LIN {X 0,Y 356.432,Z 513.307,A -85,B 0,C 180,E1 -13393.092,E2 -13393.092} C_VEL
LIN {X 0,Y 355.324,Z 522.171,A -85,B 0,C 180,E1 -13395.1,E2 -13395.1} C_VEL
LIN {X 0,Y 354.334,Z 530.476,A -85,B 0,C 180,E1 -13397.398,E2 -13397.398} C_VEL
LIN {X 0,Y 353.681,Z 537.111,A -85,B 0,C 180,E1 -13399.698,E2 -13399.698} C_VEL
LIN {X 0,Y 353.432,Z 542.27,A -85,B 0,C 180,E1 -13401.999,E2 -13401.999} C_VEL
LIN {X 0,Y 353.28,Z 546.062,A -85,B 0,C 180,E1 -13404.291,E2 -13404.291} C_VEL
LIN {X 0,Y 353.247,Z 548.565,A -85,B 0,C 180,E1 -13406.578,E2 -13406.578} C_VEL
LIN {X 0,Y 353.373,Z 549.83,A -85,B 0,C 180,E1 -13408.86,E2 -13408.86} C_VEL
LIN {X 0,Y 353.373,Z 549.828,A -85,B 0,C 180,E1 -13411.139,E2 -13411.139} C_VEL
LIN {X 0,Y 353.248,Z 548.554,A -85,B 0,C 180,E1 -13413.422,E2 -13413.422} C_VEL
LIN {X 0,Y 353.308,Z 546.046,A -85,B 0,C 180,E1 -13415.708,E2 -13415.708} C_VEL
LIN {X 0,Y 353.433,Z 542.253,A -85,B 0,C 180,E1 -13418.001,E2 -13418.001} C_VEL
LIN {X 0,Y 353.681,Z 537.089,A -85,B 0,C 180,E1 -13420.302,E2 -13420.302} C_VEL
LIN {X 0,Y 354.326,Z 530.439,A -85,B 0,C 180,E1 -13422.602,E2 -13422.602} C_VEL
LIN {X 0,Y 355.299,Z 522.123,A -85,B 0,C 180,E1 -13424.901,E2 -13424.901} C_VEL
LIN {X 0,Y 356.428,Z 513.256,A -85,B 0,C 180,E1 -13426.908,E2 -13426.908} C_VEL
LIN {X 0,Y 357.977,Z 502.598,A -85,B 0,C 180,E1 -13428.901,E2 -13428.901} C_VEL
LIN {X 0,Y 359.499,Z 491.658,A -85,B 0,C 180,E1 -13430.603,E2 -13430.603} C_VEL
LIN {X 0,Y 361.192,Z 479.725,A -85,B 0,C 180,E1 -13432.148,E2 -13432.148} C_VEL
LIN {X 0,Y 363.012,Z 466.679,A -85,B 0,C 180,E1 -13433.535,E2 -13433.535} C_VEL
LIN {X 0,Y 364.699,Z 454.014,A -85,B 0,C 180,E1 -13434.628,E2 -13434.628} C_VEL
LIN {X 0,Y 365.906,Z 442.133,A -85,B 0,C 180,E1 -13435.48,E2 -13435.48} C_VEL
LIN {X 0,Y 364.101,Z 428.944,A -85,B 0,C 180,E1 -13436.443,E2 -13436.443} C_VEL
LIN {X 0,Y 361.058,Z 413.785,A -85,B 0,C 180,E1 -13437.388,E2 -13437.388} C_VEL
LIN {X 0,Y 356.966,Z 398.611,A -85,B 0,C 180,E1 -13438.183,E2 -13438.183} C_VEL
LIN {X 0,Y 356.454,Z 396.29,A -85,B 0,C 180,E1 -13438.282,E2 -13438.282} C_VEL
LIN {X 0,Y 357.714,Z 387.602,A -85,B 0,C 180,E1 -13442.348,E2 -13442.348} C_VEL
LIN {X 0,Y 358.68,Z 381.362,A -85,B 0,C 180,E1 -13445.312,E2 -13445.312} C_VEL
LIN {X 0,Y 358.879,Z 378.763,A -85,B 0,C 180,E1 -13446.591,E2 -13446.591} C_VEL
LIN {X 0,Y 357.99,Z 373.352,A -85,B 0,C 180,E1 -13449.446,E2 -13449.446} C_VEL
LIN {X 0,Y 356.788,Z 366.727,A -85,B 0,C 180,E1 -13453.212,E2 -13453.212} C_VEL
LIN {X 0,Y 355.578,Z 360.645,A -85,B 0,C 180,E1 -13456.996,E2 -13456.996} C_VEL
LIN {X 0,Y 354.833,Z 356.903,A -85,B 0,C 180,E1 -13459.56,E2 -13459.56} C_VEL
LIN {X 0,Y 354.804,Z 356.919,A -85,B 0,C 180,E1 -13463.541,E2 -13463.541} C_VEL
LIN {X 0,Y 354.832,Z 356.914,A -85,B 0,C 180,E1 -13466.318,E2 -13466.318} C_VEL
LIN {X 0,Y 354.87,Z 356.908,A -85,B 0,C 180,E1 -13470.622,E2 -13470.622} C_VEL
LIN {X 0,Y 354.902,Z 356.902,A -85,B 0,C 180,E1 -13474.173,E2 -13474.173} C_VEL
LIN {X 0,Y 354.837,Z 356.912,A -85,B 0,C 180,E1 -13477.894,E2 -13477.894} C_VEL
LIN {X 0,Y 354.926,Z 356.897,A -85,B 0,C 180,E1 -13481.892,E2 -13481.892} C_VEL
LIN {X 0,Y 354.946,Z 356.896,A -85,B 0,C 180,E1 -13485.981,E2 -13485.981} C_VEL
LIN {X 0,Y 354.982,Z 356.889,A -85,B 0,C 180,E1 -13489.736,E2 -13489.736} C_VEL
LIN {X 0,Y 355.118,Z 356.871,A -85,B 0,C 180,E1 -13493.181,E2 -13493.181} C_VEL
LIN {X 0,Y 355.247,Z 356.854,A -85,B 0,C 180,E1 -13497.733,E2 -13497.733} C_VEL
LIN {X 0,Y 355.4,Z 356.836,A -85,B 0,C 180,E1 -13500,E2 -13500} C_VEL
LIN {X 0,Y 355.247,Z 356.859,A -85,B 0,C 180,E1 -13502.268,E2 -13502.268} C_VEL
LIN {X 0,Y 355.142,Z 356.87,A -85,B 0,C 180,E1 -13506.819,E2 -13506.819} C_VEL
LIN {X 0,Y 355.02,Z 356.886,A -85,B 0,C 180,E1 -13509.112,E2 -13509.112} C_VEL
LIN {X 0,Y 354.93,Z 356.897,A -85,B 0,C 180,E1 -13512.581,E2 -13512.581} C_VEL
LIN {X 0,Y 354.894,Z 356.902,A -85,B 0,C 180,E1 -13516.096,E2 -13516.096} C_VEL
LIN {X 0,Y 354.91,Z 356.898,A -85,B 0,C 180,E1 -13518.472,E2 -13518.472} C_VEL
LIN {X 0,Y 354.838,Z 356.911,A -85,B 0,C 180,E1 -13522.106,E2 -13522.106} C_VEL
LIN {X 0,Y 354.903,Z 356.901,A -85,B 0,C 180,E1 -13525.827,E2 -13525.827} C_VEL
LIN {X 0,Y 354.857,Z 356.904,A -85,B 0,C 180,E1 -13529.679,E2 -13529.679} C_VEL
LIN {X 0,Y 354.809,Z 356.915,A -85,B 0,C 180,E1 -13533.702,E2 -13533.702} C_VEL
LIN {X 0,Y 354.801,Z 356.916,A -85,B 0,C 180,E1 -13536.459,E2 -13536.459} C_VEL
LIN {X 0,Y 354.827,Z 356.913,A -85,B 0,C 180,E1 -13539.424,E2 -13539.424} C_VEL
LIN {X 0,Y 354.791,Z 356.916,A -85,B 0,C 180,E1 -13542.867,E2 -13542.867} C_VEL
LIN {X 0,Y 354.817,Z 357.055,A -85,B 0,C 180,E1 -13544.515,E2 -13544.515} C_VEL
LIN {X 0,Y 355.42,Z 360.567,A -85,B 0,C 180,E1 -13547.754,E2 -13547.754} C_VEL
LIN {X 0,Y 355.755,Z 364.073,A -85,B 0,C 180,E1 -13550.79,E2 -13550.79} C_VEL
LIN {X 0,Y 355.617,Z 367.534,A -85,B 0,C 180,E1 -13553.638,E2 -13553.638} C_VEL
LIN {X 0,Y 355.366,Z 371,A -85,B 0,C 180,E1 -13556.375,E2 -13556.375} C_VEL
LIN {X 0,Y 355.058,Z 374.488,A -85,B 0,C 180,E1 -13559.026,E2 -13559.026} C_VEL
LIN {X 0,Y 354.822,Z 378.006,A -85,B 0,C 180,E1 -13561.616,E2 -13561.616} C_VEL
LIN {X 0,Y 354.625,Z 381.777,A -85,B 0,C 180,E1 -13564.292,E2 -13564.292} C_VEL
LIN {X 0,Y 356.695,Z 387.842,A -85,B 0,C 180,E1 -13564.635,E2 -13564.635} C_VEL
LIN {X 0,Y 361.427,Z 402.417,A -85,B 0,C 180,E1 -13565.559,E2 -13565.559} C_VEL
LIN {X 0,Y 364.83,Z 415.964,A -85,B 0,C 180,E1 -13566.556,E2 -13566.556} C_VEL
LIN {X 0,Y 366.104,Z 422.295,A -85,B 0,C 180,E1 -13567.074,E2 -13567.074} C_VEL
LIN {X 0,Y 364.894,Z 435.031,A -85,B 0,C 180,E1 -13568.017,E2 -13568.017} C_VEL
LIN {X 0,Y 363.543,Z 446.261,A -85,B 0,C 180,E1 -13569.045,E2 -13569.045} C_VEL
LIN {X 0,Y 361.82,Z 458.433,A -85,B 0,C 180,E1 -13570.423,E2 -13570.423} C_VEL
LIN {X 0,Y 360.396,Z 468.475,A -85,B 0,C 180,E1 -13571.819,E2 -13571.819} C_VEL
LIN {X 0,Y 358.753,Z 478.455,A -85,B 0,C 180,E1 -13573.498,E2 -13573.498} C_VEL
LIN {X 0,Y 357.49,Z 486.727,A -85,B 0,C 180,E1 -13575.193,E2 -13575.193} C_VEL
LIN {X 0,Y 356.185,Z 494.631,A -85,B 0,C 180,E1 -13577.175,E2 -13577.175} C_VEL
LIN {X 0,Y 355.172,Z 501.015,A -85,B 0,C 180,E1 -13579.165,E2 -13579.165} C_VEL
LIN {X 0,Y 354.358,Z 506.684,A -85,B 0,C 180,E1 -13581.446,E2 -13581.446} C_VEL
LIN {X 0,Y 353.991,Z 509.96,A -85,B 0,C 180,E1 -13583.159,E2 -13583.159} C_VEL
LIN {X 0,Y 353.57,Z 513.105,A -85,B 0,C 180,E1 -13585.44,E2 -13585.44} C_VEL
LIN {X 0,Y 353.496,Z 514.951,A -85,B 0,C 180,E1 -13587.721,E2 -13587.721} C_VEL
LIN {X 0,Y 353.397,Z 515.581,A -85,B 0,C 180,E1 -13590,E2 -13590} C_VEL
LIN {X 0,Y 353.495,Z 515.006,A -85,B 0,C 180,E1 -13592.279,E2 -13592.279} C_VEL
LIN {X 0,Y 353.569,Z 513.22,A -85,B 0,C 180,E1 -13594.561,E2 -13594.561} C_VEL
LIN {X 0,Y 353.991,Z 510.136,A -85,B 0,C 180,E1 -13596.842,E2 -13596.842} C_VEL
LIN {X 0,Y 354.514,Z 505.659,A -85,B 0,C 180,E1 -13599.126,E2 -13599.126} C_VEL
LIN {X 0,Y 355.381,Z 499.628,A -85,B 0,C 180,E1 -13601.406,E2 -13601.406} C_VEL
LIN {X 0,Y 356.468,Z 492.907,A -85,B 0,C 180,E1 -13603.395,E2 -13603.395} C_VEL
LIN {X 0,Y 357.863,Z 484.866,A -85,B 0,C 180,E1 -13605.309,E2 -13605.309} C_VEL
LIN {X 0,Y 358.945,Z 477.477,A -85,B 0,C 180,E1 -13606.786,E2 -13606.786} C_VEL
LIN {X 0,Y 360.595,Z 467.25,A -85,B 0,C 180,E1 -13608.465,E2 -13608.465} C_VEL
LIN {X 0,Y 362.254,Z 455.812,A -85,B 0,C 180,E1 -13609.995,E2 -13609.995} C_VEL
LIN {X 0,Y 363.811,Z 444.405,A -85,B 0,C 180,E1 -13611.236,E2 -13611.236} C_VEL
LIN {X 0,Y 365.265,Z 431.504,A -85,B 0,C 180,E1 -13612.367,E2 -13612.367} C_VEL
LIN {X 0,Y 366.073,Z 421.795,A -85,B 0,C 180,E1 -13613.069,E2 -13613.069} C_VEL
LIN {X 0,Y 362.89,Z 407.718,A -85,B 0,C 180,E1 -13614.172,E2 -13614.172} C_VEL
LIN {X 0,Y 359.006,Z 394.651,A -85,B 0,C 180,E1 -13615.06,E2 -13615.06} C_VEL
LIN {X 0,Y 354.616,Z 381.77,A -85,B 0,C 180,E1 -13615.818,E2 -13615.818} C_VEL
LIN {X 0,Y 354.944,Z 376.407,A -85,B 0,C 180,E1 -13619.671,E2 -13619.671} C_VEL
LIN {X 0,Y 355.117,Z 374.097,A -85,B 0,C 180,E1 -13621.397,E2 -13621.397} C_VEL
LIN {X 0,Y 354.59,Z 372.967,A -85,B 0,C 180,E1 -13622.327,E2 -13622.327} C_VEL
LIN {X 0,Y 351.952,Z 371.428,A -85,B 0,C 180,E1 -13623.855,E2 -13623.855} C_VEL
LIN {X 0,Y 349.672,Z 370.256,A -85,B 0,C 180,E1 -13625.092,E2 -13625.092} C_VEL
LIN {X 0,Y 348.705,Z 369.259,A -85,B 0,C 180,E1 -13626.044,E2 -13626.044} C_VEL
LIN {X 0,Y 348.635,Z 368.886,A -85,B 0,C 180,E1 -13626.364,E2 -13626.364} C_VEL
LIN {X 0,Y 348.761,Z 366.131,A -85,B 0,C 180,E1 -13628.66,E2 -13628.66} C_VEL
LIN {X 0,Y 348.733,Z 364.408,A -85,B 0,C 180,E1 -13630.158,E2 -13630.158} C_VEL
LIN {X 0,Y 348.284,Z 360.78,A -85,B 0,C 180,E1 -13633.411,E2 -13633.411} C_VEL
LIN {X 0,Y 347.734,Z 357.793,A -85,B 0,C 180,E1 -13636.394,E2 -13636.394} C_VEL
LIN {X 0,Y 347.736,Z 357.792,A -85,B 0,C 180,E1 -13639.703,E2 -13639.703} C_VEL
LIN {X 0,Y 347.766,Z 357.79,A -85,B 0,C 180,E1 -13642.679,E2 -13642.679} C_VEL
LIN {X 0,Y 347.752,Z 357.791,A -85,B 0,C 180,E1 -13645.956,E2 -13645.956} C_VEL
LIN {X 0,Y 347.768,Z 357.79,A -85,B 0,C 180,E1 -13649.654,E2 -13649.654} C_VEL
LIN {X 0,Y 347.856,Z 357.78,A -85,B 0,C 180,E1 -13652.745,E2 -13652.745} C_VEL
LIN {X 0,Y 347.793,Z 357.786,A -85,B 0,C 180,E1 -13656.162,E2 -13656.162} C_VEL
LIN {X 0,Y 347.817,Z 357.783,A -85,B 0,C 180,E1 -13659.909,E2 -13659.909} C_VEL
LIN {X 0,Y 347.871,Z 357.775,A -85,B 0,C 180,E1 -13662.359,E2 -13662.359} C_VEL
LIN {X 0,Y 347.902,Z 357.773,A -85,B 0,C 180,E1 -13665.971,E2 -13665.971} C_VEL
LIN {X 0,Y 347.934,Z 357.77,A -85,B 0,C 180,E1 -13669.526,E2 -13669.526} C_VEL
LIN {X 0,Y 348.08,Z 357.748,A -85,B 0,C 180,E1 -13671.875,E2 -13671.875} C_VEL
LIN {X 0,Y 348.073,Z 357.75,A -85,B 0,C 180,E1 -13674.206,E2 -13674.206} C_VEL
LIN {X 0,Y 348.211,Z 357.732,A -85,B 0,C 180,E1 -13677.686,E2 -13677.686} C_VEL
LIN {X 0,Y 348.35,Z 357.72,A -85,B 0,C 180,E1 -13680,E2 -13680} C_VEL
LIN {X 0,Y 348.211,Z 357.735,A -85,B 0,C 180,E1 -13682.313,E2 -13682.313} C_VEL
LIN {X 0,Y 348.082,Z 357.751,A -85,B 0,C 180,E1 -13686.958,E2 -13686.958} C_VEL
LIN {X 0,Y 347.935,Z 357.768,A -85,B 0,C 180,E1 -13690.474,E2 -13690.474} C_VEL
LIN {X 0,Y 347.902,Z 357.774,A -85,B 0,C 180,E1 -13694.149,E2 -13694.149} C_VEL
LIN {X 0,Y 347.895,Z 357.78,A -85,B 0,C 180,E1 -13698.29,E2 -13698.29} C_VEL
LIN {X 0,Y 347.793,Z 357.793,A -85,B 0,C 180,E1 -13701.635,E2 -13701.635} C_VEL
LIN {X 0,Y 347.816,Z 357.784,A -85,B 0,C 180,E1 -13705.108,E2 -13705.108} C_VEL
LIN {X 0,Y 347.814,Z 357.786,A -85,B 0,C 180,E1 -13707.693,E2 -13707.693} C_VEL
LIN {X 0,Y 347.767,Z 357.79,A -85,B 0,C 180,E1 -13710.346,E2 -13710.346} C_VEL
LIN {X 0,Y 347.747,Z 357.795,A -85,B 0,C 180,E1 -13714.463,E2 -13714.463} C_VEL
LIN {X 0,Y 347.777,Z 357.793,A -85,B 0,C 180,E1 -13717.988,E2 -13717.988} C_VEL
LIN {X 0,Y 347.804,Z 357.927,A -85,B 0,C 180,E1 -13719.837,E2 -13719.837} C_VEL
LIN {X 0,Y 348.884,Z 363.299,A -85,B 0,C 180,E1 -13723.515,E2 -13723.515} C_VEL
LIN {X 0,Y 349.967,Z 368.768,A -85,B 0,C 180,E1 -13726.938,E2 -13726.938} C_VEL
LIN {X 0,Y 350.961,Z 374.276,A -85,B 0,C 180,E1 -13730.148,E2 -13730.148} C_VEL
LIN {X 0,Y 351.897,Z 379.829,A -85,B 0,C 180,E1 -13733.19,E2 -13733.19} C_VEL
LIN {X 0,Y 351.615,Z 383.488,A -85,B 0,C 180,E1 -13735.034,E2 -13735.034} C_VEL
LIN {X 0,Y 350.384,Z 390.794,A -85,B 0,C 180,E1 -13738.566,E2 -13738.566} C_VEL
LIN {X 0,Y 349.561,Z 396.09,A -85,B 0,C 180,E1 -13741.108,E2 -13741.108} C_VEL
LIN {X 0,Y 354.345,Z 414.03,A -85,B 0,C 180,E1 -13742.083,E2 -13742.083} C_VEL
LIN {X 0,Y 357.089,Z 427.45,A -85,B 0,C 180,E1 -13742.946,E2 -13742.946} C_VEL
LIN {X 0,Y 359.156,Z 441.19,A -85,B 0,C 180,E1 -13743.971,E2 -13743.971} C_VEL
LIN {X 0,Y 359.363,Z 442.934,A -85,B 0,C 180,E1 -13744.107,E2 -13744.107} C_VEL
LIN {X 0,Y 357.759,Z 457.127,A -85,B 0,C 180,E1 -13745.171,E2 -13745.171} C_VEL
LIN {X 0,Y 355.932,Z 470.571,A -85,B 0,C 180,E1 -13746.431,E2 -13746.431} C_VEL
LIN {X 0,Y 354.131,Z 482.904,A -85,B 0,C 180,E1 -13747.847,E2 -13747.847} C_VEL
LIN {X 0,Y 352.535,Z 492.979,A -85,B 0,C 180,E1 -13749.229,E2 -13749.229} C_VEL
LIN {X 0,Y 350.988,Z 503.92,A -85,B 0,C 180,E1 -13751.011,E2 -13751.011} C_VEL
LIN {X 0,Y 349.523,Z 512.923,A -85,B 0,C 180,E1 -13752.747,E2 -13752.747} C_VEL
LIN {X 0,Y 348.361,Z 521.799,A -85,B 0,C 180,E1 -13754.795,E2 -13754.795} C_VEL
LIN {X 0,Y 347.322,Z 530.113,A -85,B 0,C 180,E1 -13757.139,E2 -13757.139} C_VEL
LIN {X 0,Y 346.63,Z 536.754,A -85,B 0,C 180,E1 -13759.486,E2 -13759.486} C_VEL
LIN {X 0,Y 346.357,Z 541.918,A -85,B 0,C 180,E1 -13761.834,E2 -13761.834} C_VEL
LIN {X 0,Y 346.199,Z 545.714,A -85,B 0,C 180,E1 -13764.174,E2 -13764.174} C_VEL
LIN {X 0,Y 346.168,Z 548.22,A -85,B 0,C 180,E1 -13766.508,E2 -13766.508} C_VEL
LIN {X 0,Y 346.276,Z 549.485,A -85,B 0,C 180,E1 -13768.837,E2 -13768.837} C_VEL
LIN {X 0,Y 346.276,Z 549.482,A -85,B 0,C 180,E1 -13771.163,E2 -13771.163} C_VEL
LIN {X 0,Y 346.17,Z 548.208,A -85,B 0,C 180,E1 -13773.492,E2 -13773.492} C_VEL
LIN {X 0,Y 346.243,Z 545.52,A -85,B 0,C 180,E1 -13775.961,E2 -13775.961} C_VEL
LIN {X 0,Y 346.357,Z 541.9,A -85,B 0,C 180,E1 -13778.166,E2 -13778.166} C_VEL
LIN {X 0,Y 346.63,Z 536.73,A -85,B 0,C 180,E1 -13780.514,E2 -13780.514} C_VEL
LIN {X 0,Y 347.311,Z 530.073,A -85,B 0,C 180,E1 -13782.861,E2 -13782.861} C_VEL
LIN {X 0,Y 348.357,Z 521.749,A -85,B 0,C 180,E1 -13785.205,E2 -13785.205} C_VEL
LIN {X 0,Y 349.516,Z 512.868,A -85,B 0,C 180,E1 -13787.253,E2 -13787.253} C_VEL
LIN {X 0,Y 350.938,Z 503.85,A -85,B 0,C 180,E1 -13788.992,E2 -13788.992} C_VEL
LIN {X 0,Y 352.548,Z 492.92,A -85,B 0,C 180,E1 -13790.767,E2 -13790.767} C_VEL
LIN {X 0,Y 354.24,Z 481.636,A -85,B 0,C 180,E1 -13792.299,E2 -13792.299} C_VEL
LIN {X 0,Y 356.037,Z 469.04,A -85,B 0,C 180,E1 -13793.715,E2 -13793.715} C_VEL
LIN {X 0,Y 357.767,Z 456.972,A -85,B 0,C 180,E1 -13794.828,E2 -13794.828} C_VEL
LIN {X 0,Y 359.291,Z 443.142,A -85,B 0,C 180,E1 -13795.869,E2 -13795.869} C_VEL
LIN {X 0,Y 357.443,Z 429.698,A -85,B 0,C 180,E1 -13796.887,E2 -13796.887} C_VEL
LIN {X 0,Y 354.554,Z 414.95,A -85,B 0,C 180,E1 -13797.844,E2 -13797.844} C_VEL
LIN {X 0,Y 350.68,Z 400.439,A -85,B 0,C 180,E1 -13798.649,E2 -13798.649} C_VEL
LIN {X 0,Y 349.562,Z 396.051,A -85,B 0,C 180,E1 -13798.892,E2 -13798.892} C_VEL
LIN {X 0,Y 350.804,Z 388.028,A -85,B 0,C 180,E1 -13802.746,E2 -13802.746} C_VEL
LIN {X 0,Y 351.725,Z 382.545,A -85,B 0,C 180,E1 -13805.413,E2 -13805.413} C_VEL
LIN {X 0,Y 351.845,Z 379.503,A -85,B 0,C 180,E1 -13806.967,E2 -13806.967} C_VEL
LIN {X 0,Y 350.943,Z 374.198,A -85,B 0,C 180,E1 -13809.854,E2 -13809.854} C_VEL
LIN {X 0,Y 349.763,Z 367.681,A -85,B 0,C 180,E1 -13813.667,E2 -13813.667} C_VEL
LIN {X 0,Y 348.559,Z 361.667,A -85,B 0,C 180,E1 -13817.51,E2 -13817.51} C_VEL
LIN {X 0,Y 347.797,Z 357.79,A -85,B 0,C 180,E1 -13820.262,E2 -13820.262} C_VEL
LIN {X 0,Y 347.792,Z 357.793,A -85,B 0,C 180,E1 -13824.125,E2 -13824.125} C_VEL
LIN {X 0,Y 347.741,Z 357.797,A -85,B 0,C 180,E1 -13828.086,E2 -13828.086} C_VEL
LIN {X 0,Y 347.807,Z 357.789,A -85,B 0,C 180,E1 -13830.99,E2 -13830.99} C_VEL
LIN {X 0,Y 347.834,Z 357.784,A -85,B 0,C 180,E1 -13833.608,E2 -13833.608} C_VEL
LIN {X 0,Y 347.791,Z 357.787,A -85,B 0,C 180,E1 -13836.162,E2 -13836.162} C_VEL
LIN {X 0,Y 347.82,Z 357.786,A -85,B 0,C 180,E1 -13839.91,E2 -13839.91} C_VEL
LIN {X 0,Y 347.869,Z 357.776,A -85,B 0,C 180,E1 -13842.36,E2 -13842.36} C_VEL
LIN {X 0,Y 347.9,Z 357.774,A -85,B 0,C 180,E1 -13845.971,E2 -13845.971} C_VEL
LIN {X 0,Y 347.933,Z 357.769,A -85,B 0,C 180,E1 -13849.526,E2 -13849.526} C_VEL
LIN {X 0,Y 348.086,Z 357.748,A -85,B 0,C 180,E1 -13853.042,E2 -13853.042} C_VEL
LIN {X 0,Y 348.21,Z 357.731,A -85,B 0,C 180,E1 -13857.687,E2 -13857.687} C_VEL
LIN {X 0,Y 348.349,Z 357.714,A -85,B 0,C 180,E1 -13860,E2 -13860} C_VEL
LIN {X 0,Y 348.21,Z 357.736,A -85,B 0,C 180,E1 -13862.314,E2 -13862.314} C_VEL
LIN {X 0,Y 348.11,Z 357.745,A -85,B 0,C 180,E1 -13866.958,E2 -13866.958} C_VEL
LIN {X 0,Y 347.973,Z 357.764,A -85,B 0,C 180,E1 -13869.299,E2 -13869.299} C_VEL
LIN {X 0,Y 347.898,Z 357.774,A -85,B 0,C 180,E1 -13872.839,E2 -13872.839} C_VEL
LIN {X 0,Y 347.843,Z 357.782,A -85,B 0,C 180,E1 -13876.431,E2 -13876.431} C_VEL
LIN {X 0,Y 347.859,Z 357.779,A -85,B 0,C 180,E1 -13878.86,E2 -13878.86} C_VEL
LIN {X 0,Y 347.778,Z 357.789,A -85,B 0,C 180,E1 -13882.579,E2 -13882.579} C_VEL
LIN {X 0,Y 347.816,Z 357.784,A -85,B 0,C 180,E1 -13885.108,E2 -13885.108} C_VEL
LIN {X 0,Y 347.814,Z 357.783,A -85,B 0,C 180,E1 -13887.694,E2 -13887.694} C_VEL
LIN {X 0,Y 347.767,Z 357.79,A -85,B 0,C 180,E1 -13890.346,E2 -13890.346} C_VEL
LIN {X 0,Y 347.747,Z 357.794,A -85,B 0,C 180,E1 -13894.464,E2 -13894.464} C_VEL
LIN {X 0,Y 347.776,Z 357.79,A -85,B 0,C 180,E1 -13897.989,E2 -13897.989} C_VEL
LIN {X 0,Y 347.753,Z 357.793,A -85,B 0,C 180,E1 -13901.83,E2 -13901.83} C_VEL
LIN {X 0,Y 347.75,Z 357.918,A -85,B 0,C 180,E1 -13904.005,E2 -13904.005} C_VEL
LIN {X 0,Y 348.299,Z 360.743,A -85,B 0,C 180,E1 -13906.681,E2 -13906.681} C_VEL
LIN {X 0,Y 348.715,Z 364.377,A -85,B 0,C 180,E1 -13909.983,E2 -13909.983} C_VEL
LIN {X 0,Y 348.673,Z 367.707,A -85,B 0,C 180,E1 -13912.793,E2 -13912.793} C_VEL
LIN {X 0,Y 348.411,Z 371.417,A -85,B 0,C 180,E1 -13915.796,E2 -13915.796} C_VEL
LIN {X 0,Y 348.133,Z 374.692,A -85,B 0,C 180,E1 -13918.34,E2 -13918.34} C_VEL
LIN {X 0,Y 347.843,Z 378.22,A -85,B 0,C 180,E1 -13920.993,E2 -13920.993} C_VEL
LIN {X 0,Y 347.611,Z 381.993,A -85,B 0,C 180,E1 -13923.714,E2 -13923.714} C_VEL
LIN {X 0,Y 353.042,Z 397.77,A -85,B 0,C 180,E1 -13924.687,E2 -13924.687} C_VEL
LIN {X 0,Y 356.691,Z 410.649,A -85,B 0,C 180,E1 -13925.614,E2 -13925.614} C_VEL
LIN {X 0,Y 359.45,Z 423.04,A -85,B 0,C 180,E1 -13926.636,E2 -13926.636} C_VEL
LIN {X 0,Y 358.328,Z 435.735,A -85,B 0,C 180,E1 -13927.611,E2 -13927.611} C_VEL
LIN {X 0,Y 356.932,Z 446.729,A -85,B 0,C 180,E1 -13928.638,E2 -13928.638} C_VEL
LIN {X 0,Y 355.336,Z 457.783,A -85,B 0,C 180,E1 -13929.901,E2 -13929.901} C_VEL
LIN {X 0,Y 353.661,Z 468.878,A -85,B 0,C 180,E1 -13931.461,E2 -13931.461} C_VEL
LIN {X 0,Y 351.957,Z 478.84,A -85,B 0,C 180,E1 -13933.17,E2 -13933.17} C_VEL
LIN {X 0,Y 350.624,Z 487.1,A -85,B 0,C 180,E1 -13934.896,E2 -13934.896} C_VEL
LIN {X 0,Y 349.241,Z 494.996,A -85,B 0,C 180,E1 -13936.915,E2 -13936.915} C_VEL
LIN {X 0,Y 348.186,Z 501.372,A -85,B 0,C 180,E1 -13938.945,E2 -13938.945} C_VEL
LIN {X 0,Y 347.339,Z 507.036,A -85,B 0,C 180,E1 -13941.271,E2 -13941.271} C_VEL
LIN {X 0,Y 346.946,Z 510.311,A -85,B 0,C 180,E1 -13943.019,E2 -13943.019} C_VEL
LIN {X 0,Y 346.512,Z 513.452,A -85,B 0,C 180,E1 -13945.347,E2 -13945.347} C_VEL
LIN {X 0,Y 346.404,Z 515.297,A -85,B 0,C 180,E1 -13947.675,E2 -13947.675} C_VEL
LIN {X 0,Y 346.318,Z 515.925,A -85,B 0,C 180,E1 -13950,E2 -13950} C_VEL
LIN {X 0,Y 346.403,Z 515.352,A -85,B 0,C 180,E1 -13952.326,E2 -13952.326} C_VEL
LIN {X 0,Y 346.511,Z 513.565,A -85,B 0,C 180,E1 -13954.654,E2 -13954.654} C_VEL
LIN {X 0,Y 346.946,Z 510.484,A -85,B 0,C 180,E1 -13956.981,E2 -13956.981} C_VEL
LIN {X 0,Y 347.502,Z 506.011,A -85,B 0,C 180,E1 -13959.311,E2 -13959.311} C_VEL
LIN {X 0,Y 348.419,Z 499.985,A -85,B 0,C 180,E1 -13961.637,E2 -13961.637} C_VEL
LIN {X 0,Y 349.552,Z 493.272,A -85,B 0,C 180,E1 -13963.665,E2 -13963.665} C_VEL
LIN {X 0,Y 350.976,Z 485.438,A -85,B 0,C 180,E1 -13965.572,E2 -13965.572} C_VEL
LIN {X 0,Y 352.138,Z 477.863,A -85,B 0,C 180,E1 -13967.121,E2 -13967.121} C_VEL
LIN {X 0,Y 353.887,Z 467.657,A -85,B 0,C 180,E1 -13968.828,E2 -13968.828} C_VEL
LIN {X 0,Y 355.424,Z 457.419,A -85,B 0,C 180,E1 -13970.245,E2 -13970.245} C_VEL
LIN {X 0,Y 357.055,Z 446.3,A -85,B 0,C 180,E1 -13971.506,E2 -13971.506} C_VEL
LIN {X 0,Y 358.532,Z 433.687,A -85,B 0,C 180,E1 -13972.67,E2 -13972.67} C_VEL
LIN {X 0,Y 359.568,Z 423.86,A -85,B 0,C 180,E1 -13973.397,E2 -13973.397} C_VEL
LIN {X 0,Y 356.919,Z 411.45,A -85,B 0,C 180,E1 -13974.426,E2 -13974.426} C_VEL
LIN {X 0,Y 353.318,Z 398.651,A -85,B 0,C 180,E1 -13975.359,E2 -13975.359} C_VEL
LIN {X 0,Y 348.541,Z 384.929,A -85,B 0,C 180,E1 -13976.23,E2 -13976.23} C_VEL
LIN {X 0,Y 347.619,Z 381.964,A -85,B 0,C 180,E1 -13976.41,E2 -13976.41} C_VEL
LIN {X 0,Y 347.976,Z 376.617,A -85,B 0,C 180,E1 -13980.326,E2 -13980.326} C_VEL
LIN {X 0,Y 348.262,Z 373.108,A -85,B 0,C 180,E1 -13983.016,E2 -13983.016} C_VEL
LIN {X 0,Y 348.635,Z 368.886,A -85,B 0,C 180,E1 -13986.364,E2 -13986.364} C_VEL
LIN {X 0,Y 348.009,Z 367.867,A -85,B 0,C 180,E1 -13987.315,E2 -13987.315} C_VEL
LIN {X 0,Y 345.216,Z 366.529,A -85,B 0,C 180,E1 -13988.873,E2 -13988.873} C_VEL
LIN {X 0,Y 342.788,Z 365.501,A -85,B 0,C 180,E1 -13990.134,E2 -13990.134} C_VEL
LIN {X 0,Y 341.677,Z 364.596,A -85,B 0,C 180,E1 -13991.107,E2 -13991.107} C_VEL
LIN {X 0,Y 341.55,Z 364.255,A -85,B 0,C 180,E1 -13991.435,E2 -13991.435} C_VEL
LIN {X 0,Y 341.07,Z 361,A -85,B 0,C 180,E1 -13994.475,E2 -13994.475} C_VEL
LIN {X 0,Y 340.68,Z 358.671,A -85,B 0,C 180,E1 -13996.87,E2 -13996.87} C_VEL
LIN {X 0,Y 340.703,Z 358.668,A -85,B 0,C 180,E1 -14000.248,E2 -14000.248} C_VEL
LIN {X 0,Y 340.714,Z 358.669,A -85,B 0,C 180,E1 -14003.559,E2 -14003.559} C_VEL
LIN {X 0,Y 340.696,Z 358.671,A -85,B 0,C 180,E1 -14006.154,E2 -14006.154} C_VEL
LIN {X 0,Y 340.779,Z 358.663,A -85,B 0,C 180,E1 -14010.333,E2 -14010.333} C_VEL
LIN {X 0,Y 340.809,Z 358.66,A -85,B 0,C 180,E1 -14013.02,E2 -14013.02} C_VEL
LIN {X 0,Y 340.761,Z 358.663,A -85,B 0,C 180,E1 -14015.638,E2 -14015.638} C_VEL
LIN {X 0,Y 340.75,Z 358.66,A -85,B 0,C 180,E1 -14019.474,E2 -14019.474} C_VEL
LIN {X 0,Y 340.862,Z 358.647,A -85,B 0,C 180,E1 -14021.984,E2 -14021.984} C_VEL
LIN {X 0,Y 340.874,Z 358.648,A -85,B 0,C 180,E1 -14025.705,E2 -14025.705} C_VEL
LIN {X 0,Y 340.876,Z 358.648,A -85,B 0,C 180,E1 -14029.306,E2 -14029.306} C_VEL
LIN {X 0,Y 341.081,Z 358.623,A -85,B 0,C 180,E1 -14032.898,E2 -14032.898} C_VEL
LIN {X 0,Y 341.173,Z 358.609,A -85,B 0,C 180,E1 -14037.639,E2 -14037.639} C_VEL
LIN {X 0,Y 341.3,Z 358.598,A -85,B 0,C 180,E1 -14040,E2 -14040} C_VEL
LIN {X 0,Y 341.173,Z 358.612,A -85,B 0,C 180,E1 -14042.361,E2 -14042.361} C_VEL
LIN {X 0,Y 341.05,Z 358.626,A -85,B 0,C 180,E1 -14047.102,E2 -14047.102} C_VEL
LIN {X 0,Y 340.878,Z 358.646,A -85,B 0,C 180,E1 -14050.693,E2 -14050.693} C_VEL
LIN {X 0,Y 340.867,Z 358.65,A -85,B 0,C 180,E1 -14054.324,E2 -14054.324} C_VEL
LIN {X 0,Y 340.842,Z 358.66,A -85,B 0,C 180,E1 -14058.467,E2 -14058.467} C_VEL
LIN {X 0,Y 340.757,Z 358.667,A -85,B 0,C 180,E1 -14061.856,E2 -14061.856} C_VEL
LIN {X 0,Y 340.776,Z 358.661,A -85,B 0,C 180,E1 -14065.664,E2 -14065.664} C_VEL
LIN {X 0,Y 340.744,Z 358.667,A -85,B 0,C 180,E1 -14068.319,E2 -14068.319} C_VEL
LIN {X 0,Y 340.707,Z 358.673,A -85,B 0,C 180,E1 -14071.044,E2 -14071.044} C_VEL
LIN {X 0,Y 340.721,Z 358.675,A -85,B 0,C 180,E1 -14075.278,E2 -14075.278} C_VEL
LIN {X 0,Y 340.729,Z 358.706,A -85,B 0,C 180,E1 -14079.013,E2 -14079.013} C_VEL
LIN {X 0,Y 341.794,Z 363.925,A -85,B 0,C 180,E1 -14082.73,E2 -14082.73} C_VEL
LIN {X 0,Y 342.74,Z 368.716,A -85,B 0,C 180,E1 -14085.864,E2 -14085.864} C_VEL
LIN {X 0,Y 343.732,Z 374.131,A -85,B 0,C 180,E1 -14089.157,E2 -14089.157} C_VEL
LIN {X 0,Y 344.815,Z 380.267,A -85,B 0,C 180,E1 -14092.645,E2 -14092.645} C_VEL
LIN {X 0,Y 344.942,Z 382.387,A -85,B 0,C 180,E1 -14093.782,E2 -14093.782} C_VEL
LIN {X 0,Y 343.915,Z 388.618,A -85,B 0,C 180,E1 -14096.913,E2 -14096.913} C_VEL
LIN {X 0,Y 342.719,Z 395.923,A -85,B 0,C 180,E1 -14100.517,E2 -14100.517} C_VEL
LIN {X 0,Y 347.509,Z 413.681,A -85,B 0,C 180,E1 -14101.511,E2 -14101.511} C_VEL
LIN {X 0,Y 350.429,Z 427.822,A -85,B 0,C 180,E1 -14102.45,E2 -14102.45} C_VEL
LIN {X 0,Y 352.491,Z 441.872,A -85,B 0,C 180,E1 -14103.534,E2 -14103.534} C_VEL
LIN {X 0,Y 352.606,Z 445.116,A -85,B 0,C 180,E1 -14103.792,E2 -14103.792} C_VEL
LIN {X 0,Y 351.055,Z 458.246,A -85,B 0,C 180,E1 -14104.825,E2 -14104.825} C_VEL
LIN {X 0,Y 349.175,Z 471.414,A -85,B 0,C 180,E1 -14106.104,E2 -14106.104} C_VEL
LIN {X 0,Y 347.326,Z 483.574,A -85,B 0,C 180,E1 -14107.547,E2 -14107.547} C_VEL
LIN {X 0,Y 345.613,Z 494.023,A -85,B 0,C 180,E1 -14109.024,E2 -14109.024} C_VEL
LIN {X 0,Y 343.946,Z 505.175,A -85,B 0,C 180,E1 -14110.917,E2 -14110.917} C_VEL
LIN {X 0,Y 342.269,Z 515.293,A -85,B 0,C 180,E1 -14112.986,E2 -14112.986} C_VEL
LIN {X 0,Y 341.149,Z 523.721,A -85,B 0,C 180,E1 -14115.077,E2 -14115.077} C_VEL
LIN {X 0,Y 340.145,Z 531.602,A -85,B 0,C 180,E1 -14117.47,E2 -14117.47} C_VEL
LIN {X 0,Y 339.477,Z 537.861,A -85,B 0,C 180,E1 -14119.865,E2 -14119.865} C_VEL
LIN {X 0,Y 339.218,Z 542.677,A -85,B 0,C 180,E1 -14122.26,E2 -14122.26} C_VEL
LIN {X 0,Y 339.128,Z 545.451,A -85,B 0,C 180,E1 -14124.118,E2 -14124.118} C_VEL
LIN {X 0,Y 339.092,Z 547.874,A -85,B 0,C 180,E1 -14126.435,E2 -14126.435} C_VEL
LIN {X 0,Y 339.179,Z 549.139,A -85,B 0,C 180,E1 -14128.813,E2 -14128.813} C_VEL
LIN {X 0,Y 339.222,Z 549.303,A -85,B 0,C 180,E1 -14130,E2 -14130} C_VEL
LIN {X 0,Y 339.09,Z 548.652,A -85,B 0,C 180,E1 -14132.376,E2 -14132.376} C_VEL
LIN {X 0,Y 339.127,Z 546.763,A -85,B 0,C 180,E1 -14134.755,E2 -14134.755} C_VEL
LIN {X 0,Y 339.222,Z 543.614,A -85,B 0,C 180,E1 -14137.141,E2 -14137.141} C_VEL
LIN {X 0,Y 339.394,Z 539.137,A -85,B 0,C 180,E1 -14139.536,E2 -14139.536} C_VEL
LIN {X 0,Y 339.962,Z 533.238,A -85,B 0,C 180,E1 -14141.931,E2 -14141.931} C_VEL
LIN {X 0,Y 340.783,Z 525.762,A -85,B 0,C 180,E1 -14144.328,E2 -14144.328} C_VEL
LIN {X 0,Y 341.893,Z 517.762,A -85,B 0,C 180,E1 -14146.418,E2 -14146.418} C_VEL
LIN {X 0,Y 343.427,Z 508.15,A -85,B 0,C 180,E1 -14148.494,E2 -14148.494} C_VEL
LIN {X 0,Y 344.967,Z 498.35,A -85,B 0,C 180,E1 -14150.264,E2 -14150.264} C_VEL
LIN {X 0,Y 346.714,Z 486.705,A -85,B 0,C 180,E1 -14152.024,E2 -14152.024} C_VEL
LIN {X 0,Y 348.746,Z 473.884,A -85,B 0,C 180,E1 -14153.611,E2 -14153.611} C_VEL
LIN {X 0,Y 350.58,Z 461.209,A -85,B 0,C 180,E1 -14154.897,E2 -14154.897} C_VEL
LIN {X 0,Y 352.324,Z 447.392,A -85,B 0,C 180,E1 -14156.03,E2 -14156.03} C_VEL
LIN {X 0,Y 352.71,Z 443.953,A -85,B 0,C 180,E1 -14156.278,E2 -14156.278} C_VEL
LIN {X 0,Y 350.89,Z 430.908,A -85,B 0,C 180,E1 -14157.311,E2 -14157.311} C_VEL
LIN {X 0,Y 348.227,Z 416.81,A -85,B 0,C 180,E1 -14158.271,E2 -14158.271} C_VEL
LIN {X 0,Y 344.357,Z 401.886,A -85,B 0,C 180,E1 -14159.147,E2 -14159.147} C_VEL
LIN {X 0,Y 342.713,Z 395.88,A -85,B 0,C 180,E1 -14159.483,E2 -14159.483} C_VEL
LIN {X 0,Y 343.913,Z 388.583,A -85,B 0,C 180,E1 -14163.086,E2 -14163.086} C_VEL
LIN {X 0,Y 344.915,Z 382.337,A -85,B 0,C 180,E1 -14166.221,E2 -14166.221} C_VEL
LIN {X 0,Y 344.54,Z 378.324,A -85,B 0,C 180,E1 -14168.407,E2 -14168.407} C_VEL
LIN {X 0,Y 343.195,Z 371.255,A -85,B 0,C 180,E1 -14172.515,E2 -14172.515} C_VEL
LIN {X 0,Y 342.13,Z 365.788,A -85,B 0,C 180,E1 -14175.97,E2 -14175.97} C_VEL
LIN {X 0,Y 341.104,Z 360.436,A -85,B 0,C 180,E1 -14179.671,E2 -14179.671} C_VEL
LIN {X 0,Y 340.738,Z 358.669,A -85,B 0,C 180,E1 -14180.986,E2 -14180.986} C_VEL
LIN {X 0,Y 340.72,Z 358.675,A -85,B 0,C 180,E1 -14184.722,E2 -14184.722} C_VEL
LIN {X 0,Y 340.706,Z 358.675,A -85,B 0,C 180,E1 -14188.956,E2 -14188.956} C_VEL
LIN {X 0,Y 340.781,Z 358.661,A -85,B 0,C 180,E1 -14192.474,E2 -14192.474} C_VEL
LIN {X 0,Y 340.758,Z 358.665,A -85,B 0,C 180,E1 -14195.639,E2 -14195.639} C_VEL
LIN {X 0,Y 340.751,Z 358.662,A -85,B 0,C 180,E1 -14199.475,E2 -14199.475} C_VEL
LIN {X 0,Y 340.861,Z 358.649,A -85,B 0,C 180,E1 -14201.985,E2 -14201.985} C_VEL
LIN {X 0,Y 340.872,Z 358.649,A -85,B 0,C 180,E1 -14205.705,E2 -14205.705} C_VEL
LIN {X 0,Y 340.876,Z 358.649,A -85,B 0,C 180,E1 -14209.307,E2 -14209.307} C_VEL
LIN {X 0,Y 341.053,Z 358.625,A -85,B 0,C 180,E1 -14212.898,E2 -14212.898} C_VEL
LIN {X 0,Y 341.171,Z 358.607,A -85,B 0,C 180,E1 -14217.639,E2 -14217.639} C_VEL
LIN {X 0,Y 341.299,Z 358.592,A -85,B 0,C 180,E1 -14220,E2 -14220} C_VEL
LIN {X 0,Y 341.171,Z 358.612,A -85,B 0,C 180,E1 -14222.361,E2 -14222.361} C_VEL
LIN {X 0,Y 341.08,Z 358.62,A -85,B 0,C 180,E1 -14227.102,E2 -14227.102} C_VEL
LIN {X 0,Y 340.879,Z 358.646,A -85,B 0,C 180,E1 -14230.694,E2 -14230.694} C_VEL
LIN {X 0,Y 340.866,Z 358.648,A -85,B 0,C 180,E1 -14234.325,E2 -14234.325} C_VEL
LIN {X 0,Y 340.841,Z 358.65,A -85,B 0,C 180,E1 -14238.467,E2 -14238.467} C_VEL
LIN {X 0,Y 340.757,Z 358.662,A -85,B 0,C 180,E1 -14241.857,E2 -14241.857} C_VEL
LIN {X 0,Y 340.776,Z 358.661,A -85,B 0,C 180,E1 -14245.664,E2 -14245.664} C_VEL
LIN {X 0,Y 340.744,Z 358.667,A -85,B 0,C 180,E1 -14248.32,E2 -14248.32} C_VEL
LIN {X 0,Y 340.707,Z 358.67,A -85,B 0,C 180,E1 -14251.044,E2 -14251.044} C_VEL
LIN {X 0,Y 340.721,Z 358.671,A -85,B 0,C 180,E1 -14255.279,E2 -14255.279} C_VEL
LIN {X 0,Y 340.712,Z 358.669,A -85,B 0,C 180,E1 -14258.386,E2 -14258.386} C_VEL
LIN {X 0,Y 340.701,Z 358.673,A -85,B 0,C 180,E1 -14262.046,E2 -14262.046} C_VEL
LIN {X 0,Y 340.713,Z 358.819,A -85,B 0,C 180,E1 -14263.511,E2 -14263.511} C_VEL
LIN {X 0,Y 341.194,Z 361.508,A -85,B 0,C 180,E1 -14266.132,E2 -14266.132} C_VEL
LIN {X 0,Y 341.686,Z 365.209,A -85,B 0,C 180,E1 -14269.556,E2 -14269.556} C_VEL
LIN {X 0,Y 341.731,Z 367.878,A -85,B 0,C 180,E1 -14271.904,E2 -14271.904} C_VEL
LIN {X 0,Y 341.431,Z 372.128,A -85,B 0,C 180,E1 -14275.423,E2 -14275.423} C_VEL
LIN {X 0,Y 341.013,Z 376.658,A -85,B 0,C 180,E1 -14278.987,E2 -14278.987} C_VEL
LIN {X 0,Y 340.685,Z 381.346,A -85,B 0,C 180,E1 -14282.505,E2 -14282.505} C_VEL
LIN {X 0,Y 340.655,Z 382.153,A -85,B 0,C 180,E1 -14283.099,E2 -14283.099} C_VEL
LIN {X 0,Y 341.735,Z 385.452,A -85,B 0,C 180,E1 -14283.291,E2 -14283.291} C_VEL
LIN {X 0,Y 346.616,Z 399.446,A -85,B 0,C 180,E1 -14284.217,E2 -14284.217} C_VEL
LIN {X 0,Y 350.183,Z 412.204,A -85,B 0,C 180,E1 -14285.182,E2 -14285.182} C_VEL
LIN {X 0,Y 352.749,Z 423.844,A -85,B 0,C 180,E1 -14286.181,E2 -14286.181} C_VEL
LIN {X 0,Y 352.771,Z 426.742,A -85,B 0,C 180,E1 -14286.409,E2 -14286.409} C_VEL
LIN {X 0,Y 351.3,Z 440.313,A -85,B 0,C 180,E1 -14287.534,E2 -14287.534} C_VEL
LIN {X 0,Y 349.693,Z 452.352,A -85,B 0,C 180,E1 -14288.792,E2 -14288.792} C_VEL
LIN {X 0,Y 347.88,Z 463.525,A -85,B 0,C 180,E1 -14290.221,E2 -14290.221} C_VEL
LIN {X 0,Y 346.019,Z 474.488,A -85,B 0,C 180,E1 -14291.956,E2 -14291.956} C_VEL
LIN {X 0,Y 344.365,Z 483.752,A -85,B 0,C 180,E1 -14293.753,E2 -14293.753} C_VEL
LIN {X 0,Y 342.94,Z 492.164,A -85,B 0,C 180,E1 -14295.764,E2 -14295.764} C_VEL
LIN {X 0,Y 341.851,Z 498.276,A -85,B 0,C 180,E1 -14297.534,E2 -14297.534} C_VEL
LIN {X 0,Y 340.735,Z 504.755,A -85,B 0,C 180,E1 -14299.903,E2 -14299.903} C_VEL
LIN {X 0,Y 340.013,Z 509.643,A -85,B 0,C 180,E1 -14302.279,E2 -14302.279} C_VEL
LIN {X 0,Y 339.68,Z 512.395,A -85,B 0,C 180,E1 -14304.062,E2 -14304.062} C_VEL
LIN {X 0,Y 339.328,Z 514.879,A -85,B 0,C 180,E1 -14306.438,E2 -14306.438} C_VEL
LIN {X 0,Y 339.274,Z 516.107,A -85,B 0,C 180,E1 -14308.813,E2 -14308.813} C_VEL
LIN {X 0,Y 339.274,Z 516.133,A -85,B 0,C 180,E1 -14311.187,E2 -14311.187} C_VEL
LIN {X 0,Y 339.327,Z 514.961,A -85,B 0,C 180,E1 -14313.563,E2 -14313.563} C_VEL
LIN {X 0,Y 339.679,Z 512.536,A -85,B 0,C 180,E1 -14315.938,E2 -14315.938} C_VEL
LIN {X 0,Y 340.147,Z 508.782,A -85,B 0,C 180,E1 -14318.316,E2 -14318.316} C_VEL
LIN {X 0,Y 340.949,Z 503.557,A -85,B 0,C 180,E1 -14320.692,E2 -14320.692} C_VEL
LIN {X 0,Y 342.071,Z 496.685,A -85,B 0,C 180,E1 -14323.062,E2 -14323.062} C_VEL
LIN {X 0,Y 343.542,Z 489.09,A -85,B 0,C 180,E1 -14325.12,E2 -14325.12} C_VEL
LIN {X 0,Y 344.863,Z 481.184,A -85,B 0,C 180,E1 -14326.882,E2 -14326.882} C_VEL
LIN {X 0,Y 346.543,Z 471.648,A -85,B 0,C 180,E1 -14328.628,E2 -14328.628} C_VEL
LIN {X 0,Y 348.275,Z 461.067,A -85,B 0,C 180,E1 -14330.217,E2 -14330.217} C_VEL
LIN {X 0,Y 350.102,Z 449.355,A -85,B 0,C 180,E1 -14331.646,E2 -14331.646} C_VEL
LIN {X 0,Y 351.745,Z 436.776,A -85,B 0,C 180,E1 -14332.886,E2 -14332.886} C_VEL
LIN {X 0,Y 352.93,Z 424.653,A -85,B 0,C 180,E1 -14333.848,E2 -14333.848} C_VEL
LIN {X 0,Y 350.239,Z 412.156,A -85,B 0,C 180,E1 -14334.923,E2 -14334.923} C_VEL
LIN {X 0,Y 346.503,Z 398.991,A -85,B 0,C 180,E1 -14335.92,E2 -14335.92} C_VEL
LIN {X 0,Y 341.671,Z 385.294,A -85,B 0,C 180,E1 -14336.828,E2 -14336.828} C_VEL
LIN {X 0,Y 340.657,Z 382.132,A -85,B 0,C 180,E1 -14337.024,E2 -14337.024} C_VEL
LIN {X 0,Y 340.938,Z 378.092,A -85,B 0,C 180,E1 -14340.028,E2 -14340.028} C_VEL
LIN {X 0,Y 341.326,Z 373.3,A -85,B 0,C 180,E1 -14343.776,E2 -14343.776} C_VEL
LIN {X 0,Y 341.672,Z 369.733,A -85,B 0,C 180,E1 -14346.658,E2 -14346.658} C_VEL
LIN {X 0,Y 341.761,Z 366.302,A -85,B 0,C 180,E1 -14349.605,E2 -14349.605} C_VEL
LIN {X 0,Y 341.55,Z 364.255,A -85,B 0,C 180,E1 -14351.435,E2 -14351.435} C_VEL
LIN {X 0,Y 340.746,Z 363.346,A -85,B 0,C 180,E1 -14352.405,E2 -14352.405} C_VEL
LIN {X 0,Y 337.676,Z 362.218,A -85,B 0,C 180,E1 -14353.985,E2 -14353.985} C_VEL
LIN {X 0,Y 335.078,Z 361.372,A -85,B 0,C 180,E1 -14355.266,E2 -14355.266} C_VEL
LIN {X 0,Y 333.888,Z 360.581,A -85,B 0,C 180,E1 -14356.257,E2 -14356.257} C_VEL
LIN {X 0,Y 333.749,Z 360.266,A -85,B 0,C 180,E1 -14356.593,E2 -14356.593} C_VEL
LIN {X 0,Y 333.644,Z 359.547,A -85,B 0,C 180,E1 -14357.618,E2 -14357.618} C_VEL
LIN {X 0,Y 333.656,Z 359.546,A -85,B 0,C 180,E1 -14361.202,E2 -14361.202} C_VEL
LIN {X 0,Y 333.68,Z 359.545,A -85,B 0,C 180,E1 -14363.861,E2 -14363.861} C_VEL
LIN {X 0,Y 333.647,Z 359.549,A -85,B 0,C 180,E1 -14367.413,E2 -14367.413} C_VEL
LIN {X 0,Y 333.715,Z 359.542,A -85,B 0,C 180,E1 -14371.028,E2 -14371.028} C_VEL
LIN {X 0,Y 333.74,Z 359.535,A -85,B 0,C 180,E1 -14373.754,E2 -14373.754} C_VEL
LIN {X 0,Y 333.724,Z 359.541,A -85,B 0,C 180,E1 -14377.914,E2 -14377.914} C_VEL
LIN {X 0,Y 333.798,Z 359.528,A -85,B 0,C 180,E1 -14381.589,E2 -14381.589} C_VEL
LIN {X 0,Y 333.813,Z 359.527,A -85,B 0,C 180,E1 -14385.576,E2 -14385.576} C_VEL
LIN {X 0,Y 333.839,Z 359.525,A -85,B 0,C 180,E1 -14389.078,E2 -14389.078} C_VEL
LIN {X 0,Y 334.031,Z 359.501,A -85,B 0,C 180,E1 -14392.747,E2 -14392.747} C_VEL
LIN {X 0,Y 333.815,Z 359.524,A -85,B 0,C 180,E1 -14395.169,E2 -14395.169} C_VEL
LIN {X 0,Y 334.11,Z 359.489,A -85,B 0,C 180,E1 -14397.589,E2 -14397.589} C_VEL
LIN {X 0,Y 334.251,Z 359.477,A -85,B 0,C 180,E1 -14400,E2 -14400} C_VEL
LIN {X 0,Y 334.11,Z 359.492,A -85,B 0,C 180,E1 -14402.411,E2 -14402.411} C_VEL
LIN {X 0,Y 334.013,Z 359.504,A -85,B 0,C 180,E1 -14406.039,E2 -14406.039} C_VEL
LIN {X 0,Y 333.854,Z 359.526,A -85,B 0,C 180,E1 -14409.695,E2 -14409.695} C_VEL
LIN {X 0,Y 333.803,Z 359.532,A -85,B 0,C 180,E1 -14413.391,E2 -14413.391} C_VEL
LIN {X 0,Y 333.751,Z 359.538,A -85,B 0,C 180,E1 -14417.146,E2 -14417.146} C_VEL
LIN {X 0,Y 333.746,Z 359.538,A -85,B 0,C 180,E1 -14419.69,E2 -14419.69} C_VEL
LIN {X 0,Y 333.696,Z 359.543,A -85,B 0,C 180,E1 -14422.278,E2 -14422.278} C_VEL
LIN {X 0,Y 333.739,Z 359.54,A -85,B 0,C 180,E1 -14426.246,E2 -14426.246} C_VEL
LIN {X 0,Y 333.714,Z 359.543,A -85,B 0,C 180,E1 -14428.972,E2 -14428.972} C_VEL
LIN {X 0,Y 333.648,Z 359.551,A -85,B 0,C 180,E1 -14432.587,E2 -14432.587} C_VEL
LIN {X 0,Y 333.679,Z 359.551,A -85,B 0,C 180,E1 -14436.138,E2 -14436.138} C_VEL
LIN {X 0,Y 333.716,Z 359.598,A -85,B 0,C 180,E1 -14438.248,E2 -14438.248} C_VEL
LIN {X 0,Y 334.769,Z 364.961,A -85,B 0,C 180,E1 -14442.206,E2 -14442.206} C_VEL
LIN {X 0,Y 335.714,Z 369.642,A -85,B 0,C 180,E1 -14445.379,E2 -14445.379} C_VEL
LIN {X 0,Y 336.677,Z 374.979,A -85,B 0,C 180,E1 -14448.719,E2 -14448.719} C_VEL
LIN {X 0,Y 337.766,Z 381.018,A -85,B 0,C 180,E1 -14452.249,E2 -14452.249} C_VEL
LIN {X 0,Y 337.852,Z 384.61,A -85,B 0,C 180,E1 -14454.221,E2 -14454.221} C_VEL
LIN {X 0,Y 336.595,Z 391.689,A -85,B 0,C 180,E1 -14457.83,E2 -14457.83} C_VEL
LIN {X 0,Y 335.873,Z 395.952,A -85,B 0,C 180,E1 -14459.91,E2 -14459.91} C_VEL
LIN {X 0,Y 340.314,Z 411.998,A -85,B 0,C 180,E1 -14460.829,E2 -14460.829} C_VEL
LIN {X 0,Y 343.522,Z 426.734,A -85,B 0,C 180,E1 -14461.832,E2 -14461.832} C_VEL
LIN {X 0,Y 345.671,Z 441.133,A -85,B 0,C 180,E1 -14462.963,E2 -14462.963} C_VEL
LIN {X 0,Y 346.023,Z 446.004,A -85,B 0,C 180,E1 -14463.375,E2 -14463.375} C_VEL
LIN {X 0,Y 344.361,Z 459.458,A -85,B 0,C 180,E1 -14464.477,E2 -14464.477} C_VEL
LIN {X 0,Y 342.413,Z 472.25,A -85,B 0,C 180,E1 -14465.763,E2 -14465.763} C_VEL
LIN {X 0,Y 340.519,Z 484.225,A -85,B 0,C 180,E1 -14467.233,E2 -14467.233} C_VEL
LIN {X 0,Y 338.734,Z 494.778,A -85,B 0,C 180,E1 -14468.774,E2 -14468.774} C_VEL
LIN {X 0,Y 337.166,Z 504.783,A -85,B 0,C 180,E1 -14470.518,E2 -14470.518} C_VEL
LIN {X 0,Y 335.4,Z 514.917,A -85,B 0,C 180,E1 -14472.626,E2 -14472.626} C_VEL
LIN {X 0,Y 334.179,Z 523.35,A -85,B 0,C 180,E1 -14474.759,E2 -14474.759} C_VEL
LIN {X 0,Y 333.32,Z 529.388,A -85,B 0,C 180,E1 -14476.589,E2 -14476.589} C_VEL
LIN {X 0,Y 332.543,Z 536.041,A -85,B 0,C 180,E1 -14479.035,E2 -14479.035} C_VEL
LIN {X 0,Y 332.212,Z 541.214,A -85,B 0,C 180,E1 -14481.484,E2 -14481.484} C_VEL
LIN {X 0,Y 332.04,Z 545.018,A -85,B 0,C 180,E1 -14483.925,E2 -14483.925} C_VEL
LIN {X 0,Y 332.016,Z 547.529,A -85,B 0,C 180,E1 -14486.359,E2 -14486.359} C_VEL
LIN {X 0,Y 332.082,Z 548.794,A -85,B 0,C 180,E1 -14488.787,E2 -14488.787} C_VEL
LIN {X 0,Y 332.13,Z 548.958,A -85,B 0,C 180,E1 -14490,E2 -14490} C_VEL
LIN {X 0,Y 332.001,Z 548.306,A -85,B 0,C 180,E1 -14492.426,E2 -14492.426} C_VEL
LIN {X 0,Y 332.031,Z 546.415,A -85,B 0,C 180,E1 -14494.857,E2 -14494.857} C_VEL
LIN {X 0,Y 332.137,Z 543.262,A -85,B 0,C 180,E1 -14497.294,E2 -14497.294} C_VEL
LIN {X 0,Y 332.333,Z 538.781,A -85,B 0,C 180,E1 -14499.74,E2 -14499.74} C_VEL
LIN {X 0,Y 332.95,Z 532.877,A -85,B 0,C 180,E1 -14502.186,E2 -14502.186} C_VEL
LIN {X 0,Y 333.856,Z 525.396,A -85,B 0,C 180,E1 -14504.632,E2 -14504.632} C_VEL
LIN {X 0,Y 334.986,Z 517.383,A -85,B 0,C 180,E1 -14506.767,E2 -14506.767} C_VEL
LIN {X 0,Y 336.621,Z 507.76,A -85,B 0,C 180,E1 -14508.881,E2 -14508.881} C_VEL
LIN {X 0,Y 338.326,Z 497.212,A -85,B 0,C 180,E1 -14510.808,E2 -14510.808} C_VEL
LIN {X 0,Y 340.257,Z 485.2,A -85,B 0,C 180,E1 -14512.625,E2 -14512.625} C_VEL
LIN {X 0,Y 342.344,Z 472.127,A -85,B 0,C 180,E1 -14514.241,E2 -14514.241} C_VEL
LIN {X 0,Y 344.323,Z 459.306,A -85,B 0,C 180,E1 -14515.525,E2 -14515.525} C_VEL
LIN {X 0,Y 345.891,Z 446.819,A -85,B 0,C 180,E1 -14516.552,E2 -14516.552} C_VEL
LIN {X 0,Y 346.101,Z 444.973,A -85,B 0,C 180,E1 -14516.687,E2 -14516.687} C_VEL
LIN {X 0,Y 344.224,Z 430.976,A -85,B 0,C 180,E1 -14517.835,E2 -14517.835} C_VEL
LIN {X 0,Y 341.358,Z 416.367,A -85,B 0,C 180,E1 -14518.869,E2 -14518.869} C_VEL
LIN {X 0,Y 337.591,Z 401.958,A -85,B 0,C 180,E1 -14519.746,E2 -14519.746} C_VEL
LIN {X 0,Y 335.832,Z 395.772,A -85,B 0,C 180,E1 -14520.088,E2 -14520.088} C_VEL
LIN {X 0,Y 337.05,Z 389.061,A -85,B 0,C 180,E1 -14523.482,E2 -14523.482} C_VEL
LIN {X 0,Y 337.948,Z 383.501,A -85,B 0,C 180,E1 -14526.352,E2 -14526.352} C_VEL
LIN {X 0,Y 337.509,Z 379.385,A -85,B 0,C 180,E1 -14528.66,E2 -14528.66} C_VEL
LIN {X 0,Y 336.175,Z 372.16,A -85,B 0,C 180,E1 -14532.971,E2 -14532.971} C_VEL
LIN {X 0,Y 335.192,Z 367.162,A -85,B 0,C 180,E1 -14536.218,E2 -14536.218} C_VEL
LIN {X 0,Y 334.16,Z 361.733,A -85,B 0,C 180,E1 -14540.099,E2 -14540.099} C_VEL
LIN {X 0,Y 333.697,Z 359.547,A -85,B 0,C 180,E1 -14541.749,E2 -14541.749} C_VEL
LIN {X 0,Y 333.676,Z 359.552,A -85,B 0,C 180,E1 -14545.342,E2 -14545.342} C_VEL
LIN {X 0,Y 333.704,Z 359.546,A -85,B 0,C 180,E1 -14549.711,E2 -14549.711} C_VEL
LIN {X 0,Y 333.745,Z 359.537,A -85,B 0,C 180,E1 -14552.402,E2 -14552.402} C_VEL
LIN {X 0,Y 333.729,Z 359.541,A -85,B 0,C 180,E1 -14555.091,E2 -14555.091} C_VEL
LIN {X 0,Y 333.684,Z 359.54,A -85,B 0,C 180,E1 -14559.02,E2 -14559.02} C_VEL
LIN {X 0,Y 333.797,Z 359.527,A -85,B 0,C 180,E1 -14561.59,E2 -14561.59} C_VEL
LIN {X 0,Y 333.811,Z 359.528,A -85,B 0,C 180,E1 -14565.577,E2 -14565.577} C_VEL
LIN {X 0,Y 333.839,Z 359.525,A -85,B 0,C 180,E1 -14569.078,E2 -14569.078} C_VEL
LIN {X 0,Y 333.999,Z 359.505,A -85,B 0,C 180,E1 -14572.747,E2 -14572.747} C_VEL
LIN {X 0,Y 333.812,Z 359.531,A -85,B 0,C 180,E1 -14575.169,E2 -14575.169} C_VEL
LIN {X 0,Y 334.109,Z 359.487,A -85,B 0,C 180,E1 -14577.589,E2 -14577.589} C_VEL
LIN {X 0,Y 334.25,Z 359.469,A -85,B 0,C 180,E1 -14580,E2 -14580} C_VEL
LIN {X 0,Y 334.109,Z 359.492,A -85,B 0,C 180,E1 -14582.411,E2 -14582.411} C_VEL
LIN {X 0,Y 334.03,Z 359.497,A -85,B 0,C 180,E1 -14587.253,E2 -14587.253} C_VEL
LIN {X 0,Y 333.841,Z 359.522,A -85,B 0,C 180,E1 -14590.922,E2 -14590.922} C_VEL
LIN {X 0,Y 333.812,Z 359.525,A -85,B 0,C 180,E1 -14594.634,E2 -14594.634} C_VEL
LIN {X 0,Y 333.8,Z 359.528,A -85,B 0,C 180,E1 -14598.656,E2 -14598.656} C_VEL
LIN {X 0,Y 333.695,Z 359.544,A -85,B 0,C 180,E1 -14602.278,E2 -14602.278} C_VEL
LIN {X 0,Y 333.739,Z 359.538,A -85,B 0,C 180,E1 -14606.246,E2 -14606.246} C_VEL
LIN {X 0,Y 333.714,Z 359.538,A -85,B 0,C 180,E1 -14608.972,E2 -14608.972} C_VEL
LIN {X 0,Y 333.646,Z 359.549,A -85,B 0,C 180,E1 -14612.587,E2 -14612.587} C_VEL
LIN {X 0,Y 333.679,Z 359.546,A -85,B 0,C 180,E1 -14616.139,E2 -14616.139} C_VEL
LIN {X 0,Y 333.649,Z 359.552,A -85,B 0,C 180,E1 -14619.192,E2 -14619.192} C_VEL
LIN {X 0,Y 333.645,Z 359.562,A -85,B 0,C 180,E1 -14622.806,E2 -14622.806} C_VEL
LIN {X 0,Y 334.222,Z 362.815,A -85,B 0,C 180,E1 -14626.058,E2 -14626.058} C_VEL
LIN {X 0,Y 334.689,Z 366.338,A -85,B 0,C 180,E1 -14629.386,E2 -14629.386} C_VEL
LIN {X 0,Y 334.774,Z 368.069,A -85,B 0,C 180,E1 -14630.965,E2 -14630.965} C_VEL
LIN {X 0,Y 334.555,Z 371.572,A -85,B 0,C 180,E1 -14633.971,E2 -14633.971} C_VEL
LIN {X 0,Y 334.238,Z 375.587,A -85,B 0,C 180,E1 -14637.255,E2 -14637.255} C_VEL
LIN {X 0,Y 333.792,Z 380.466,A -85,B 0,C 180,E1 -14641.036,E2 -14641.036} C_VEL
LIN {X 0,Y 333.67,Z 382.319,A -85,B 0,C 180,E1 -14642.431,E2 -14642.431} C_VEL
LIN {X 0,Y 334.702,Z 385.493,A -85,B 0,C 180,E1 -14642.643,E2 -14642.643} C_VEL
LIN {X 0,Y 339.651,Z 399.279,A -85,B 0,C 180,E1 -14643.596,E2 -14643.596} C_VEL
LIN {X 0,Y 343.26,Z 411.852,A -85,B 0,C 180,E1 -14644.578,E2 -14644.578} C_VEL
LIN {X 0,Y 346.297,Z 425.744,A -85,B 0,C 180,E1 -14645.815,E2 -14645.815} C_VEL
LIN {X 0,Y 345.114,Z 438.448,A -85,B 0,C 180,E1 -14646.873,E2 -14646.873} C_VEL
LIN {X 0,Y 343.46,Z 450.232,A -85,B 0,C 180,E1 -14648.072,E2 -14648.072} C_VEL
LIN {X 0,Y 341.506,Z 461.839,A -85,B 0,C 180,E1 -14649.522,E2 -14649.522} C_VEL
LIN {X 0,Y 339.921,Z 471.445,A -85,B 0,C 180,E1 -14650.996,E2 -14650.996} C_VEL
LIN {X 0,Y 338.143,Z 481.067,A -85,B 0,C 180,E1 -14652.772,E2 -14652.772} C_VEL
LIN {X 0,Y 336.707,Z 489.047,A -85,B 0,C 180,E1 -14654.566,E2 -14654.566} C_VEL
LIN {X 0,Y 335.21,Z 496.702,A -85,B 0,C 180,E1 -14656.666,E2 -14656.666} C_VEL
LIN {X 0,Y 334.007,Z 503.643,A -85,B 0,C 180,E1 -14659.084,E2 -14659.084} C_VEL
LIN {X 0,Y 333.144,Z 508.931,A -85,B 0,C 180,E1 -14661.508,E2 -14661.508} C_VEL
LIN {X 0,Y 332.624,Z 512.744,A -85,B 0,C 180,E1 -14663.936,E2 -14663.936} C_VEL
LIN {X 0,Y 332.251,Z 515.225,A -85,B 0,C 180,E1 -14666.362,E2 -14666.362} C_VEL
LIN {X 0,Y 332.183,Z 516.452,A -85,B 0,C 180,E1 -14668.788,E2 -14668.788} C_VEL
LIN {X 0,Y 332.183,Z 516.478,A -85,B 0,C 180,E1 -14671.212,E2 -14671.212} C_VEL
LIN {X 0,Y 332.249,Z 515.306,A -85,B 0,C 180,E1 -14673.639,E2 -14673.639} C_VEL
LIN {X 0,Y 332.622,Z 512.882,A -85,B 0,C 180,E1 -14676.065,E2 -14676.065} C_VEL
LIN {X 0,Y 333.136,Z 509.13,A -85,B 0,C 180,E1 -14678.492,E2 -14678.492} C_VEL
LIN {X 0,Y 333.965,Z 503.91,A -85,B 0,C 180,E1 -14680.918,E2 -14680.918} C_VEL
LIN {X 0,Y 334.837,Z 498.943,A -85,B 0,C 180,E1 -14682.732,E2 -14682.732} C_VEL
LIN {X 0,Y 336.281,Z 491.813,A -85,B 0,C 180,E1 -14684.834,E2 -14684.834} C_VEL
LIN {X 0,Y 337.797,Z 483.021,A -85,B 0,C 180,E1 -14686.935,E2 -14686.935} C_VEL
LIN {X 0,Y 339.502,Z 473.804,A -85,B 0,C 180,E1 -14688.715,E2 -14688.715} C_VEL
LIN {X 0,Y 341.275,Z 463.61,A -85,B 0,C 180,E1 -14690.336,E2 -14690.336} C_VEL
LIN {X 0,Y 343.188,Z 452.386,A -85,B 0,C 180,E1 -14691.788,E2 -14691.788} C_VEL
LIN {X 0,Y 344.952,Z 439.712,A -85,B 0,C 180,E1 -14693.12,E2 -14693.12} C_VEL
LIN {X 0,Y 346.342,Z 427.762,A -85,B 0,C 180,E1 -14694.128,E2 -14694.128} C_VEL
LIN {X 0,Y 346.237,Z 425.458,A -85,B 0,C 180,E1 -14694.321,E2 -14694.321} C_VEL
LIN {X 0,Y 343.539,Z 412.864,A -85,B 0,C 180,E1 -14695.443,E2 -14695.443} C_VEL
LIN {X 0,Y 339.791,Z 399.709,A -85,B 0,C 180,E1 -14696.481,E2 -14696.481} C_VEL
LIN {X 0,Y 335.089,Z 386.465,A -85,B 0,C 180,E1 -14697.405,E2 -14697.405} C_VEL
LIN {X 0,Y 333.671,Z 382.333,A -85,B 0,C 180,E1 -14697.668,E2 -14697.668} C_VEL
LIN {X 0,Y 333.933,Z 378.773,A -85,B 0,C 180,E1 -14700.357,E2 -14700.357} C_VEL
LIN {X 0,Y 334.243,Z 375.276,A -85,B 0,C 180,E1 -14703.141,E2 -14703.141} C_VEL
LIN {X 0,Y 334.569,Z 371.723,A -85,B 0,C 180,E1 -14706.028,E2 -14706.028} C_VEL
LIN {X 0,Y 334.775,Z 368.206,A -85,B 0,C 180,E1 -14709.036,E2 -14709.036} C_VEL
LIN {X 0,Y 334.476,Z 364.695,A -85,B 0,C 180,E1 -14712.252,E2 -14712.252} C_VEL
LIN {X 0,Y 333.927,Z 361.157,A -85,B 0,C 180,E1 -14715.692,E2 -14715.692} C_VEL
LIN {X 0,Y 333.749,Z 360.266,A -85,B 0,C 180,E1 -14716.593,E2 -14716.593} C_VEL
LIN {X 0,Y 333.342,Z 359.821,A -85,B 0,C 180,E1 -14717.259,E2 -14717.259} C_VEL
LIN {X 0,Y 331.941,Z 359.759,A -85,B 0,C 180,E1 -14718.249,E2 -14718.249} C_VEL
LIN {X 0,Y 327.698,Z 360.302,A -85,B 0,C 180,E1 -14720.561,E2 -14720.561} C_VEL
LIN {X 0,Y 326.688,Z 360.414,A -85,B 0,C 180,E1 -14721.592,E2 -14721.592} C_VEL
LIN {X 0,Y 326.606,Z 360.422,A -85,B 0,C 180,E1 -14721.94,E2 -14721.94} C_VEL
LIN {X 0,Y 326.611,Z 360.425,A -85,B 0,C 180,E1 -14725.981,E2 -14725.981} C_VEL
LIN {X 0,Y 326.665,Z 360.421,A -85,B 0,C 180,E1 -14730.341,E2 -14730.341} C_VEL
LIN {X 0,Y 326.695,Z 360.413,A -85,B 0,C 180,E1 -14734.516,E2 -14734.516} C_VEL
LIN {X 0,Y 326.65,Z 360.418,A -85,B 0,C 180,E1 -14738.545,E2 -14738.545} C_VEL
LIN {X 0,Y 326.749,Z 360.409,A -85,B 0,C 180,E1 -14741.178,E2 -14741.178} C_VEL
LIN {X 0,Y 326.768,Z 360.403,A -85,B 0,C 180,E1 -14745.433,E2 -14745.433} C_VEL
LIN {X 0,Y 326.775,Z 360.404,A -85,B 0,C 180,E1 -14748.839,E2 -14748.839} C_VEL
LIN {X 0,Y 326.985,Z 360.379,A -85,B 0,C 180,E1 -14752.59,E2 -14752.59} C_VEL
LIN {X 0,Y 326.782,Z 360.4,A -85,B 0,C 180,E1 -14755.065,E2 -14755.065} C_VEL
LIN {X 0,Y 327.051,Z 360.368,A -85,B 0,C 180,E1 -14757.537,E2 -14757.537} C_VEL
LIN {X 0,Y 327.202,Z 360.355,A -85,B 0,C 180,E1 -14760,E2 -14760} C_VEL
LIN {X 0,Y 327.05,Z 360.371,A -85,B 0,C 180,E1 -14762.463,E2 -14762.463} C_VEL
LIN {X 0,Y 326.987,Z 360.38,A -85,B 0,C 180,E1 -14766.169,E2 -14766.169} C_VEL
LIN {X 0,Y 326.81,Z 360.405,A -85,B 0,C 180,E1 -14769.906,E2 -14769.906} C_VEL
LIN {X 0,Y 326.765,Z 360.407,A -85,B 0,C 180,E1 -14773.685,E2 -14773.685} C_VEL
LIN {X 0,Y 326.704,Z 360.417,A -85,B 0,C 180,E1 -14777.527,E2 -14777.527} C_VEL
LIN {X 0,Y 326.672,Z 360.419,A -85,B 0,C 180,E1 -14780.134,E2 -14780.134} C_VEL
LIN {X 0,Y 326.656,Z 360.423,A -85,B 0,C 180,E1 -14784.128,E2 -14784.128} C_VEL
LIN {X 0,Y 326.688,Z 360.418,A -85,B 0,C 180,E1 -14786.857,E2 -14786.857} C_VEL
LIN {X 0,Y 326.642,Z 360.423,A -85,B 0,C 180,E1 -14790.611,E2 -14790.611} C_VEL
LIN {X 0,Y 326.61,Z 360.428,A -85,B 0,C 180,E1 -14794.019,E2 -14794.019} C_VEL
LIN {X 0,Y 326.636,Z 360.579,A -85,B 0,C 180,E1 -14797.494,E2 -14797.494} C_VEL
LIN {X 0,Y 327.679,Z 365.605,A -85,B 0,C 180,E1 -14801.351,E2 -14801.351} C_VEL
LIN {X 0,Y 328.744,Z 371.002,A -85,B 0,C 180,E1 -14805.131,E2 -14805.131} C_VEL
LIN {X 0,Y 329.764,Z 376.468,A -85,B 0,C 180,E1 -14808.648,E2 -14808.648} C_VEL
LIN {X 0,Y 330.734,Z 381.96,A -85,B 0,C 180,E1 -14811.957,E2 -14811.957} C_VEL
LIN {X 0,Y 330.965,Z 385.199,A -85,B 0,C 180,E1 -14813.796,E2 -14813.796} C_VEL
LIN {X 0,Y 329.589,Z 392.784,A -85,B 0,C 180,E1 -14817.785,E2 -14817.785} C_VEL
LIN {X 0,Y 329.061,Z 395.767,A -85,B 0,C 180,E1 -14819.257,E2 -14819.257} C_VEL
LIN {X 0,Y 333.614,Z 412.049,A -85,B 0,C 180,E1 -14820.229,E2 -14820.229} C_VEL
LIN {X 0,Y 336.968,Z 427.38,A -85,B 0,C 180,E1 -14821.314,E2 -14821.314} C_VEL
LIN {X 0,Y 339.07,Z 441.753,A -85,B 0,C 180,E1 -14822.485,E2 -14822.485} C_VEL
LIN {X 0,Y 339.522,Z 446.46,A -85,B 0,C 180,E1 -14822.909,E2 -14822.909} C_VEL
LIN {X 0,Y 337.709,Z 460.371,A -85,B 0,C 180,E1 -14824.085,E2 -14824.085} C_VEL
LIN {X 0,Y 335.687,Z 473.089,A -85,B 0,C 180,E1 -14825.411,E2 -14825.411} C_VEL
LIN {X 0,Y 333.724,Z 484.878,A -85,B 0,C 180,E1 -14826.906,E2 -14826.906} C_VEL
LIN {X 0,Y 331.795,Z 495.82,A -85,B 0,C 180,E1 -14828.568,E2 -14828.568} C_VEL
LIN {X 0,Y 330.118,Z 505.934,A -85,B 0,C 180,E1 -14830.408,E2 -14830.408} C_VEL
LIN {X 0,Y 328.329,Z 515.809,A -85,B 0,C 180,E1 -14832.562,E2 -14832.562} C_VEL
LIN {X 0,Y 327.074,Z 524.046,A -85,B 0,C 180,E1 -14834.738,E2 -14834.738} C_VEL
LIN {X 0,Y 326.102,Z 530.881,A -85,B 0,C 180,E1 -14836.921,E2 -14836.921} C_VEL
LIN {X 0,Y 325.362,Z 537.151,A -85,B 0,C 180,E1 -14839.42,E2 -14839.42} C_VEL
LIN {X 0,Y 325.064,Z 541.975,A -85,B 0,C 180,E1 -14841.921,E2 -14841.921} C_VEL
LIN {X 0,Y 324.952,Z 545.168,A -85,B 0,C 180,E1 -14844.198,E2 -14844.198} C_VEL
LIN {X 0,Y 324.941,Z 547.184,A -85,B 0,C 180,E1 -14846.28,E2 -14846.28} C_VEL
LIN {X 0,Y 324.985,Z 548.448,A -85,B 0,C 180,E1 -14848.761,E2 -14848.761} C_VEL
LIN {X 0,Y 325.038,Z 548.612,A -85,B 0,C 180,E1 -14850,E2 -14850} C_VEL
LIN {X 0,Y 324.915,Z 547.961,A -85,B 0,C 180,E1 -14852.479,E2 -14852.479} C_VEL
LIN {X 0,Y 324.939,Z 546.067,A -85,B 0,C 180,E1 -14854.963,E2 -14854.963} C_VEL
LIN {X 0,Y 325.037,Z 542.91,A -85,B 0,C 180,E1 -14857.454,E2 -14857.454} C_VEL
LIN {X 0,Y 325.286,Z 538.426,A -85,B 0,C 180,E1 -14859.953,E2 -14859.953} C_VEL
LIN {X 0,Y 325.922,Z 532.516,A -85,B 0,C 180,E1 -14862.453,E2 -14862.453} C_VEL
LIN {X 0,Y 326.916,Z 525.028,A -85,B 0,C 180,E1 -14864.95,E2 -14864.95} C_VEL
LIN {X 0,Y 328.114,Z 517.006,A -85,B 0,C 180,E1 -14867.129,E2 -14867.129} C_VEL
LIN {X 0,Y 329.817,Z 507.37,A -85,B 0,C 180,E1 -14869.286,E2 -14869.286} C_VEL
LIN {X 0,Y 331.494,Z 497.535,A -85,B 0,C 180,E1 -14871.126,E2 -14871.126} C_VEL
LIN {X 0,Y 333.451,Z 485.846,A -85,B 0,C 180,E1 -14872.949,E2 -14872.949} C_VEL
LIN {X 0,Y 335.613,Z 472.959,A -85,B 0,C 180,E1 -14874.595,E2 -14874.595} C_VEL
LIN {X 0,Y 337.672,Z 460.2,A -85,B 0,C 180,E1 -14875.917,E2 -14875.917} C_VEL
LIN {X 0,Y 339.37,Z 447.452,A -85,B 0,C 180,E1 -14877.001,E2 -14877.001} C_VEL
LIN {X 0,Y 339.304,Z 443.961,A -85,B 0,C 180,E1 -14877.3,E2 -14877.3} C_VEL
LIN {X 0,Y 337.223,Z 429.233,A -85,B 0,C 180,E1 -14878.53,E2 -14878.53} C_VEL
LIN {X 0,Y 334.347,Z 415.108,A -85,B 0,C 180,E1 -14879.547,E2 -14879.547} C_VEL
LIN {X 0,Y 330.388,Z 400.634,A -85,B 0,C 180,E1 -14880.457,E2 -14880.457} C_VEL
LIN {X 0,Y 329.037,Z 395.53,A -85,B 0,C 180,E1 -14880.765,E2 -14880.765} C_VEL
LIN {X 0,Y 330.318,Z 388.588,A -85,B 0,C 180,E1 -14884.393,E2 -14884.393} C_VEL
LIN {X 0,Y 330.981,Z 384.661,A -85,B 0,C 180,E1 -14886.481,E2 -14886.481} C_VEL
LIN {X 0,Y 330.508,Z 380.54,A -85,B 0,C 180,E1 -14888.85,E2 -14888.85} C_VEL
LIN {X 0,Y 329.39,Z 374.579,A -85,B 0,C 180,E1 -14892.488,E2 -14892.488} C_VEL
LIN {X 0,Y 328.406,Z 369.35,A -85,B 0,C 180,E1 -14895.933,E2 -14895.933} C_VEL
LIN {X 0,Y 327.678,Z 365.563,A -85,B 0,C 180,E1 -14898.649,E2 -14898.649} C_VEL
LIN {X 0,Y 326.719,Z 360.961,A -85,B 0,C 180,E1 -14902.148,E2 -14902.148} C_VEL
LIN {X 0,Y 326.632,Z 360.428,A -85,B 0,C 180,E1 -14902.761,E2 -14902.761} C_VEL
LIN {X 0,Y 326.609,Z 360.43,A -85,B 0,C 180,E1 -14905.981,E2 -14905.981} C_VEL
LIN {X 0,Y 326.662,Z 360.421,A -85,B 0,C 180,E1 -14910.341,E2 -14910.341} C_VEL
LIN {X 0,Y 326.692,Z 360.415,A -85,B 0,C 180,E1 -14914.517,E2 -14914.517} C_VEL
LIN {X 0,Y 326.649,Z 360.417,A -85,B 0,C 180,E1 -14918.546,E2 -14918.546} C_VEL
LIN {X 0,Y 326.747,Z 360.405,A -85,B 0,C 180,E1 -14921.178,E2 -14921.178} C_VEL
LIN {X 0,Y 326.766,Z 360.406,A -85,B 0,C 180,E1 -14925.433,E2 -14925.433} C_VEL
LIN {X 0,Y 326.775,Z 360.405,A -85,B 0,C 180,E1 -14928.839,E2 -14928.839} C_VEL
LIN {X 0,Y 326.948,Z 360.384,A -85,B 0,C 180,E1 -14932.59,E2 -14932.59} C_VEL
LIN {X 0,Y 326.988,Z 360.374,A -85,B 0,C 180,E1 -14933.831,E2 -14933.831} C_VEL
LIN {X 0,Y 327.049,Z 360.366,A -85,B 0,C 180,E1 -14937.537,E2 -14937.537} C_VEL
LIN {X 0,Y 327.201,Z 360.347,A -85,B 0,C 180,E1 -14940,E2 -14940} C_VEL
LIN {X 0,Y 327.049,Z 360.372,A -85,B 0,C 180,E1 -14942.463,E2 -14942.463} C_VEL
LIN {X 0,Y 326.975,Z 360.377,A -85,B 0,C 180,E1 -14946.679,E2 -14946.679} C_VEL
LIN {X 0,Y 326.819,Z 360.402,A -85,B 0,C 180,E1 -14949.906,E2 -14949.906} C_VEL
LIN {X 0,Y 326.764,Z 360.406,A -85,B 0,C 180,E1 -14953.685,E2 -14953.685} C_VEL
LIN {X 0,Y 326.703,Z 360.412,A -85,B 0,C 180,E1 -14957.528,E2 -14957.528} C_VEL
LIN {X 0,Y 326.668,Z 360.419,A -85,B 0,C 180,E1 -14960.135,E2 -14960.135} C_VEL
LIN {X 0,Y 326.655,Z 360.415,A -85,B 0,C 180,E1 -14964.129,E2 -14964.129} C_VEL
LIN {X 0,Y 326.688,Z 360.412,A -85,B 0,C 180,E1 -14966.858,E2 -14966.858} C_VEL
LIN {X 0,Y 326.642,Z 360.423,A -85,B 0,C 180,E1 -14970.611,E2 -14970.611} C_VEL
LIN {X 0,Y 326.61,Z 360.428,A -85,B 0,C 180,E1 -14974.019,E2 -14974.019} C_VEL
LIN {X 0,Y 326.63,Z 360.426,A -85,B 0,C 180,E1 -14977.239,E2 -14977.239} C_VEL
LIN {X 0,Y 326.58,Z 360.431,A -85,B 0,C 180,E1 -14981.131,E2 -14981.131} C_VEL
LIN {X 0,Y 326.643,Z 360.645,A -85,B 0,C 180,E1 -14982.422,E2 -14982.422} C_VEL
LIN {X 0,Y 327.103,Z 363.282,A -85,B 0,C 180,E1 -14985.156,E2 -14985.156} C_VEL
LIN {X 0,Y 327.602,Z 366.876,A -85,B 0,C 180,E1 -14988.665,E2 -14988.665} C_VEL
LIN {X 0,Y 327.725,Z 370.004,A -85,B 0,C 180,E1 -14991.545,E2 -14991.545} C_VEL
LIN {X 0,Y 327.501,Z 373.585,A -85,B 0,C 180,E1 -14994.633,E2 -14994.633} C_VEL
LIN {X 0,Y 327.166,Z 377.089,A -85,B 0,C 180,E1 -14997.518,E2 -14997.518} C_VEL
LIN {X 0,Y 326.835,Z 380.697,A -85,B 0,C 180,E1 -15000.358,E2 -15000.358} C_VEL
LIN {X 0,Y 326.69,Z 382.529,A -85,B 0,C 180,E1 -15001.778,E2 -15001.778} C_VEL
LIN {X 0,Y 327.753,Z 385.721,A -85,B 0,C 180,E1 -15001.976,E2 -15001.976} C_VEL
LIN {X 0,Y 332.806,Z 399.482,A -85,B 0,C 180,E1 -15002.975,E2 -15002.975} C_VEL
LIN {X 0,Y 336.443,Z 411.898,A -85,B 0,C 180,E1 -15003.981,E2 -15003.981} C_VEL
LIN {X 0,Y 339.406,Z 425.434,A -85,B 0,C 180,E1 -15005.215,E2 -15005.215} C_VEL
LIN {X 0,Y 339.794,Z 427.353,A -85,B 0,C 180,E1 -15005.405,E2 -15005.405} C_VEL
LIN {X 0,Y 338.384,Z 440.317,A -85,B 0,C 180,E1 -15006.524,E2 -15006.524} C_VEL
LIN {X 0,Y 336.722,Z 451.982,A -85,B 0,C 180,E1 -15007.771,E2 -15007.771} C_VEL
LIN {X 0,Y 334.695,Z 463.327,A -85,B 0,C 180,E1 -15009.247,E2 -15009.247} C_VEL
LIN {X 0,Y 332.886,Z 473.611,A -85,B 0,C 180,E1 -15010.899,E2 -15010.899} C_VEL
LIN {X 0,Y 330.958,Z 483.612,A -85,B 0,C 180,E1 -15012.862,E2 -15012.862} C_VEL
LIN {X 0,Y 329.466,Z 491.803,A -85,B 0,C 180,E1 -15014.852,E2 -15014.852} C_VEL
LIN {X 0,Y 327.972,Z 498.995,A -85,B 0,C 180,E1 -15016.997,E2 -15016.997} C_VEL
LIN {X 0,Y 326.766,Z 505.461,A -85,B 0,C 180,E1 -15019.466,E2 -15019.466} C_VEL
LIN {X 0,Y 325.94,Z 510.343,A -85,B 0,C 180,E1 -15021.943,E2 -15021.943} C_VEL
LIN {X 0,Y 325.572,Z 513.092,A -85,B 0,C 180,E1 -15023.804,E2 -15023.804} C_VEL
LIN {X 0,Y 325.177,Z 515.571,A -85,B 0,C 180,E1 -15026.283,E2 -15026.283} C_VEL
LIN {X 0,Y 325.092,Z 516.798,A -85,B 0,C 180,E1 -15028.761,E2 -15028.761} C_VEL
LIN {X 0,Y 325.092,Z 516.823,A -85,B 0,C 180,E1 -15031.239,E2 -15031.239} C_VEL
LIN {X 0,Y 325.176,Z 515.651,A -85,B 0,C 180,E1 -15033.718,E2 -15033.718} C_VEL
LIN {X 0,Y 325.57,Z 513.228,A -85,B 0,C 180,E1 -15036.196,E2 -15036.196} C_VEL
LIN {X 0,Y 326.109,Z 509.48,A -85,B 0,C 180,E1 -15038.677,E2 -15038.677} C_VEL
LIN {X 0,Y 326.981,Z 504.264,A -85,B 0,C 180,E1 -15041.154,E2 -15041.154} C_VEL
LIN {X 0,Y 327.899,Z 499.299,A -85,B 0,C 180,E1 -15043.006,E2 -15043.006} C_VEL
LIN {X 0,Y 329.431,Z 492.174,A -85,B 0,C 180,E1 -15045.15,E2 -15045.15} C_VEL
LIN {X 0,Y 331,Z 483.397,A -85,B 0,C 180,E1 -15047.293,E2 -15047.293} C_VEL
LIN {X 0,Y 332.809,Z 474.194,A -85,B 0,C 180,E1 -15049.106,E2 -15049.106} C_VEL
LIN {X 0,Y 334.643,Z 464.022,A -85,B 0,C 180,E1 -15050.757,E2 -15050.757} C_VEL
LIN {X 0,Y 336.622,Z 452.831,A -85,B 0,C 180,E1 -15052.236,E2 -15052.236} C_VEL
LIN {X 0,Y 338.438,Z 440.331,A -85,B 0,C 180,E1 -15053.579,E2 -15053.579} C_VEL
LIN {X 0,Y 339.905,Z 428.426,A -85,B 0,C 180,E1 -15054.607,E2 -15054.607} C_VEL
LIN {X 0,Y 337.414,Z 415.74,A -85,B 0,C 180,E1 -15055.798,E2 -15055.798} C_VEL
LIN {X 0,Y 333.507,Z 401.7,A -85,B 0,C 180,E1 -15056.969,E2 -15056.969} C_VEL
LIN {X 0,Y 328.742,Z 388.185,A -85,B 0,C 180,E1 -15057.97,E2 -15057.97} C_VEL
LIN {X 0,Y 326.803,Z 383.098,A -85,B 0,C 180,E1 -15058.305,E2 -15058.305} C_VEL
LIN {X 0,Y 326.698,Z 382.487,A -85,B 0,C 180,E1 -15058.365,E2 -15058.365} C_VEL
LIN {X 0,Y 326.982,Z 379.017,A -85,B 0,C 180,E1 -15061.054,E2 -15061.054} C_VEL
LIN {X 0,Y 327.318,Z 375.477,A -85,B 0,C 180,E1 -15063.936,E2 -15063.936} C_VEL
LIN {X 0,Y 327.719,Z 371.239,A -85,B 0,C 180,E1 -15067.488,E2 -15067.488} C_VEL
LIN {X 0,Y 327.724,Z 368.403,A -85,B 0,C 180,E1 -15070.042,E2 -15070.042} C_VEL
LIN {X 0,Y 327.355,Z 364.877,A -85,B 0,C 180,E1 -15073.395,E2 -15073.395} C_VEL
LIN {X 0,Y 326.648,Z 360.755,A -85,B 0,C 180,E1 -15077.575,E2 -15077.575} C_VEL
LIN {X 0,Y 326.579,Z 360.426,A -85,B 0,C 180,E1 -15078.154,E2 -15078.154} C_VEL
LIN {X 0,Y 326.606,Z 360.422,A -85,B 0,C 180,E1 -15081.94,E2 -15081.94} C_VEL
LIN {X 0,Y 325.941,Z 360.509,A -85,B 0,C 180,E1 -15082.969,E2 -15082.969} C_VEL
LIN {X 0,Y 323.094,Z 360.865,A -85,B 0,C 180,E1 -15084.644,E2 -15084.644} C_VEL
LIN {X 0,Y 320.674,Z 361.166,A -85,B 0,C 180,E1 -15086.001,E2 -15086.001} C_VEL
LIN {X 0,Y 319.624,Z 361.297,A -85,B 0,C 180,E1 -15087.051,E2 -15087.051} C_VEL
LIN {X 0,Y 319.533,Z 361.306,A -85,B 0,C 180,E1 -15087.407,E2 -15087.407} C_VEL
LIN {X 0,Y 319.594,Z 361.301,A -85,B 0,C 180,E1 -15091.067,E2 -15091.067} C_VEL
LIN {X 0,Y 319.639,Z 361.292,A -85,B 0,C 180,E1 -15094.354,E2 -15094.354} C_VEL
LIN {X 0,Y 319.601,Z 361.301,A -85,B 0,C 180,E1 -15098.048,E2 -15098.048} C_VEL
LIN {X 0,Y 319.693,Z 361.288,A -85,B 0,C 180,E1 -15100.962,E2 -15100.962} C_VEL
LIN {X 0,Y 319.735,Z 361.279,A -85,B 0,C 180,E1 -15105.276,E2 -15105.276} C_VEL
LIN {X 0,Y 319.763,Z 361.281,A -85,B 0,C 180,E1 -15109.873,E2 -15109.873} C_VEL
LIN {X 0,Y 319.939,Z 361.257,A -85,B 0,C 180,E1 -15112.426,E2 -15112.426} C_VEL
LIN {X 0,Y 319.752,Z 361.275,A -85,B 0,C 180,E1 -15114.956,E2 -15114.956} C_VEL
LIN {X 0,Y 319.995,Z 361.247,A -85,B 0,C 180,E1 -15117.482,E2 -15117.482} C_VEL
LIN {X 0,Y 320.154,Z 361.232,A -85,B 0,C 180,E1 -15120,E2 -15120} C_VEL
LIN {X 0,Y 319.994,Z 361.25,A -85,B 0,C 180,E1 -15122.517,E2 -15122.517} C_VEL
LIN {X 0,Y 319.94,Z 361.258,A -85,B 0,C 180,E1 -15126.305,E2 -15126.305} C_VEL
LIN {X 0,Y 319.757,Z 361.281,A -85,B 0,C 180,E1 -15130.127,E2 -15130.127} C_VEL
LIN {X 0,Y 319.735,Z 361.284,A -85,B 0,C 180,E1 -15134.724,E2 -15134.724} C_VEL
LIN {X 0,Y 319.693,Z 361.291,A -85,B 0,C 180,E1 -15139.038,E2 -15139.038} C_VEL
LIN {X 0,Y 319.574,Z 361.304,A -85,B 0,C 180,E1 -15143.319,E2 -15143.319} C_VEL
LIN {X 0,Y 319.638,Z 361.296,A -85,B 0,C 180,E1 -15146.088,E2 -15146.088} C_VEL
LIN {X 0,Y 319.593,Z 361.302,A -85,B 0,C 180,E1 -15148.933,E2 -15148.933} C_VEL
LIN {X 0,Y 319.536,Z 361.308,A -85,B 0,C 180,E1 -15151.861,E2 -15151.861} C_VEL
LIN {X 0,Y 319.583,Z 361.307,A -85,B 0,C 180,E1 -15155.543,E2 -15155.543} C_VEL
LIN {X 0,Y 319.576,Z 361.42,A -85,B 0,C 180,E1 -15156.592,E2 -15156.592} C_VEL
LIN {X 0,Y 320.408,Z 365.426,A -85,B 0,C 180,E1 -15159.851,E2 -15159.851} C_VEL
LIN {X 0,Y 321.192,Z 369.282,A -85,B 0,C 180,E1 -15162.712,E2 -15162.712} C_VEL
LIN {X 0,Y 322.321,Z 375.146,A -85,B 0,C 180,E1 -15166.773,E2 -15166.773} C_VEL
LIN {X 0,Y 323.325,Z 380.641,A -85,B 0,C 180,E1 -15170.271,E2 -15170.271} C_VEL
LIN {X 0,Y 324.024,Z 385.807,A -85,B 0,C 180,E1 -15173.371,E2 -15173.371} C_VEL
LIN {X 0,Y 323.053,Z 391.319,A -85,B 0,C 180,E1 -15176.362,E2 -15176.362} C_VEL
LIN {X 0,Y 322.231,Z 395.429,A -85,B 0,C 180,E1 -15178.562,E2 -15178.562} C_VEL
LIN {X 0,Y 326.95,Z 412.142,A -85,B 0,C 180,E1 -15179.605,E2 -15179.605} C_VEL
LIN {X 0,Y 330.023,Z 426.238,A -85,B 0,C 180,E1 -15180.633,E2 -15180.633} C_VEL
LIN {X 0,Y 332.165,Z 439.936,A -85,B 0,C 180,E1 -15181.775,E2 -15181.775} C_VEL
LIN {X 0,Y 332.959,Z 447.151,A -85,B 0,C 180,E1 -15182.439,E2 -15182.439} C_VEL
LIN {X 0,Y 331.289,Z 459.876,A -85,B 0,C 180,E1 -15183.545,E2 -15183.545} C_VEL
LIN {X 0,Y 329.188,Z 472.637,A -85,B 0,C 180,E1 -15184.892,E2 -15184.892} C_VEL
LIN {X 0,Y 327.101,Z 484.454,A -85,B 0,C 180,E1 -15186.411,E2 -15186.411} C_VEL
LIN {X 0,Y 325.095,Z 495.418,A -85,B 0,C 180,E1 -15188.104,E2 -15188.104} C_VEL
LIN {X 0,Y 323.359,Z 505.55,A -85,B 0,C 180,E1 -15189.982,E2 -15189.982} C_VEL
LIN {X 0,Y 321.47,Z 515.436,A -85,B 0,C 180,E1 -15192.177,E2 -15192.177} C_VEL
LIN {X 0,Y 320.135,Z 523.681,A -85,B 0,C 180,E1 -15194.399,E2 -15194.399} C_VEL
LIN {X 0,Y 319.107,Z 530.521,A -85,B 0,C 180,E1 -15196.629,E2 -15196.629} C_VEL
LIN {X 0,Y 318.321,Z 536.797,A -85,B 0,C 180,E1 -15199.183,E2 -15199.183} C_VEL
LIN {X 0,Y 318.001,Z 541.624,A -85,B 0,C 180,E1 -15201.74,E2 -15201.74} C_VEL
LIN {X 0,Y 317.849,Z 545.059,A -85,B 0,C 180,E1 -15204.267,E2 -15204.267} C_VEL
LIN {X 0,Y 317.867,Z 546.839,A -85,B 0,C 180,E1 -15206.197,E2 -15206.197} C_VEL
LIN {X 0,Y 317.889,Z 548.103,A -85,B 0,C 180,E1 -15208.733,E2 -15208.733} C_VEL
LIN {X 0,Y 317.946,Z 548.267,A -85,B 0,C 180,E1 -15210,E2 -15210} C_VEL
LIN {X 0,Y 317.832,Z 547.615,A -85,B 0,C 180,E1 -15212.535,E2 -15212.535} C_VEL
LIN {X 0,Y 317.853,Z 545.72,A -85,B 0,C 180,E1 -15215.074,E2 -15215.074} C_VEL
LIN {X 0,Y 317.958,Z 542.56,A -85,B 0,C 180,E1 -15217.621,E2 -15217.621} C_VEL
LIN {X 0,Y 318.225,Z 538.07,A -85,B 0,C 180,E1 -15220.176,E2 -15220.176} C_VEL
LIN {X 0,Y 318.89,Z 532.154,A -85,B 0,C 180,E1 -15222.732,E2 -15222.732} C_VEL
LIN {X 0,Y 319.974,Z 524.661,A -85,B 0,C 180,E1 -15225.282,E2 -15225.282} C_VEL
LIN {X 0,Y 321.248,Z 516.629,A -85,B 0,C 180,E1 -15227.506,E2 -15227.506} C_VEL
LIN {X 0,Y 323.021,Z 506.98,A -85,B 0,C 180,E1 -15229.709,E2 -15229.709} C_VEL
LIN {X 0,Y 324.804,Z 497.129,A -85,B 0,C 180,E1 -15231.583,E2 -15231.583} C_VEL
LIN {X 0,Y 326.869,Z 485.419,A -85,B 0,C 180,E1 -15233.439,E2 -15233.439} C_VEL
LIN {X 0,Y 329.098,Z 472.498,A -85,B 0,C 180,E1 -15235.115,E2 -15235.115} C_VEL
LIN {X 0,Y 331.449,Z 458.606,A -85,B 0,C 180,E1 -15236.559,E2 -15236.559} C_VEL
LIN {X 0,Y 332.948,Z 446.975,A -85,B 0,C 180,E1 -15237.557,E2 -15237.557} C_VEL
LIN {X 0,Y 331.25,Z 433.647,A -85,B 0,C 180,E1 -15238.753,E2 -15238.753} C_VEL
LIN {X 0,Y 328.573,Z 419.061,A -85,B 0,C 180,E1 -15239.886,E2 -15239.886} C_VEL
LIN {X 0,Y 324.812,Z 404.367,A -85,B 0,C 180,E1 -15240.885,E2 -15240.885} C_VEL
LIN {X 0,Y 322.211,Z 395.382,A -85,B 0,C 180,E1 -15241.439,E2 -15241.439} C_VEL
LIN {X 0,Y 323.6,Z 388.488,A -85,B 0,C 180,E1 -15245.137,E2 -15245.137} C_VEL
LIN {X 0,Y 324.015,Z 385.773,A -85,B 0,C 180,E1 -15246.627,E2 -15246.627} C_VEL
LIN {X 0,Y 323.509,Z 381.695,A -85,B 0,C 180,E1 -15249.051,E2 -15249.051} C_VEL
LIN {X 0,Y 322.294,Z 375.076,A -85,B 0,C 180,E1 -15253.227,E2 -15253.227} C_VEL
LIN {X 0,Y 321.185,Z 369.241,A -85,B 0,C 180,E1 -15257.287,E2 -15257.287} C_VEL
LIN {X 0,Y 320.351,Z 364.906,A -85,B 0,C 180,E1 -15260.49,E2 -15260.49} C_VEL
LIN {X 0,Y 319.562,Z 361.31,A -85,B 0,C 180,E1 -15263.573,E2 -15263.573} C_VEL
LIN {X 0,Y 319.579,Z 361.306,A -85,B 0,C 180,E1 -15266.687,E2 -15266.687} C_VEL
LIN {X 0,Y 319.593,Z 361.304,A -85,B 0,C 180,E1 -15269.617,E2 -15269.617} C_VEL
LIN {X 0,Y 319.61,Z 361.298,A -85,B 0,C 180,E1 -15272.499,E2 -15272.499} C_VEL
LIN {X 0,Y 319.607,Z 361.3,A -85,B 0,C 180,E1 -15275.304,E2 -15275.304} C_VEL
LIN {X 0,Y 319.599,Z 361.299,A -85,B 0,C 180,E1 -15278.048,E2 -15278.048} C_VEL
LIN {X 0,Y 319.692,Z 361.285,A -85,B 0,C 180,E1 -15280.962,E2 -15280.962} C_VEL
LIN {X 0,Y 319.734,Z 361.282,A -85,B 0,C 180,E1 -15285.276,E2 -15285.276} C_VEL
LIN {X 0,Y 319.756,Z 361.275,A -85,B 0,C 180,E1 -15289.873,E2 -15289.873} C_VEL
LIN {X 0,Y 319.941,Z 361.251,A -85,B 0,C 180,E1 -15293.695,E2 -15293.695} C_VEL
LIN {X 0,Y 319.993,Z 361.245,A -85,B 0,C 180,E1 -15297.483,E2 -15297.483} C_VEL
LIN {X 0,Y 320.153,Z 361.225,A -85,B 0,C 180,E1 -15300,E2 -15300} C_VEL
LIN {X 0,Y 319.993,Z 361.251,A -85,B 0,C 180,E1 -15302.518,E2 -15302.518} C_VEL
LIN {X 0,Y 319.934,Z 361.255,A -85,B 0,C 180,E1 -15306.67,E2 -15306.67} C_VEL
LIN {X 0,Y 319.763,Z 361.279,A -85,B 0,C 180,E1 -15310.127,E2 -15310.127} C_VEL
LIN {X 0,Y 319.734,Z 361.277,A -85,B 0,C 180,E1 -15314.724,E2 -15314.724} C_VEL
LIN {X 0,Y 319.693,Z 361.288,A -85,B 0,C 180,E1 -15319.038,E2 -15319.038} C_VEL
LIN {X 0,Y 319.573,Z 361.301,A -85,B 0,C 180,E1 -15323.319,E2 -15323.319} C_VEL
LIN {X 0,Y 319.638,Z 361.294,A -85,B 0,C 180,E1 -15326.088,E2 -15326.088} C_VEL
LIN {X 0,Y 319.592,Z 361.298,A -85,B 0,C 180,E1 -15328.934,E2 -15328.934} C_VEL
LIN {X 0,Y 319.535,Z 361.309,A -85,B 0,C 180,E1 -15331.862,E2 -15331.862} C_VEL
LIN {X 0,Y 319.583,Z 361.303,A -85,B 0,C 180,E1 -15335.543,E2 -15335.543} C_VEL
LIN {X 0,Y 319.561,Z 361.305,A -85,B 0,C 180,E1 -15339.669,E2 -15339.669} C_VEL
LIN {X 0,Y 319.554,Z 361.353,A -85,B 0,C 180,E1 -15341.602,E2 -15341.602} C_VEL
LIN {X 0,Y 320.198,Z 364.928,A -85,B 0,C 180,E1 -15345.383,E2 -15345.383} C_VEL
LIN {X 0,Y 320.638,Z 368.449,A -85,B 0,C 180,E1 -15348.885,E2 -15348.885} C_VEL
LIN {X 0,Y 320.787,Z 370.198,A -85,B 0,C 180,E1 -15350.554,E2 -15350.554} C_VEL
LIN {X 0,Y 320.567,Z 373.741,A -85,B 0,C 180,E1 -15353.705,E2 -15353.705} C_VEL
LIN {X 0,Y 320.247,Z 377.303,A -85,B 0,C 180,E1 -15356.726,E2 -15356.726} C_VEL
LIN {X 0,Y 319.766,Z 382.291,A -85,B 0,C 180,E1 -15360.724,E2 -15360.724} C_VEL
LIN {X 0,Y 319.735,Z 382.719,A -85,B 0,C 180,E1 -15361.058,E2 -15361.058} C_VEL
LIN {X 0,Y 320.955,Z 386.144,A -85,B 0,C 180,E1 -15361.297,E2 -15361.297} C_VEL
LIN {X 0,Y 326.056,Z 399.978,A -85,B 0,C 180,E1 -15362.346,E2 -15362.346} C_VEL
LIN {X 0,Y 329.927,Z 413.223,A -85,B 0,C 180,E1 -15363.467,E2 -15363.467} C_VEL
LIN {X 0,Y 332.795,Z 426.261,A -85,B 0,C 180,E1 -15364.708,E2 -15364.708} C_VEL
LIN {X 0,Y 333.232,Z 430.093,A -85,B 0,C 180,E1 -15365.079,E2 -15365.079} C_VEL
LIN {X 0,Y 331.578,Z 442.955,A -85,B 0,C 180,E1 -15366.252,E2 -15366.252} C_VEL
LIN {X 0,Y 329.785,Z 454.861,A -85,B 0,C 180,E1 -15367.609,E2 -15367.609} C_VEL
LIN {X 0,Y 327.923,Z 464.77,A -85,B 0,C 180,E1 -15368.962,E2 -15368.962} C_VEL
LIN {X 0,Y 325.865,Z 475.661,A -85,B 0,C 180,E1 -15370.798,E2 -15370.798} C_VEL
LIN {X 0,Y 324.12,Z 484.312,A -85,B 0,C 180,E1 -15372.567,E2 -15372.567} C_VEL
LIN {X 0,Y 322.618,Z 492.169,A -85,B 0,C 180,E1 -15374.523,E2 -15374.523} C_VEL
LIN {X 0,Y 321.041,Z 499.353,A -85,B 0,C 180,E1 -15376.711,E2 -15376.711} C_VEL
LIN {X 0,Y 319.775,Z 505.815,A -85,B 0,C 180,E1 -15379.233,E2 -15379.233} C_VEL
LIN {X 0,Y 318.902,Z 510.693,A -85,B 0,C 180,E1 -15381.764,E2 -15381.764} C_VEL
LIN {X 0,Y 318.525,Z 513.44,A -85,B 0,C 180,E1 -15383.666,E2 -15383.666} C_VEL
LIN {X 0,Y 318.107,Z 515.917,A -85,B 0,C 180,E1 -15386.2,E2 -15386.2} C_VEL
LIN {X 0,Y 318.001,Z 517.143,A -85,B 0,C 180,E1 -15388.734,E2 -15388.734} C_VEL
LIN {X 0,Y 318.001,Z 517.168,A -85,B 0,C 180,E1 -15391.267,E2 -15391.267} C_VEL
LIN {X 0,Y 318.106,Z 515.996,A -85,B 0,C 180,E1 -15393.801,E2 -15393.801} C_VEL
LIN {X 0,Y 318.52,Z 513.574,A -85,B 0,C 180,E1 -15396.334,E2 -15396.334} C_VEL
LIN {X 0,Y 319.104,Z 509.828,A -85,B 0,C 180,E1 -15398.869,E2 -15398.869} C_VEL
LIN {X 0,Y 320.017,Z 504.617,A -85,B 0,C 180,E1 -15401.4,E2 -15401.4} C_VEL
LIN {X 0,Y 320.977,Z 499.654,A -85,B 0,C 180,E1 -15403.292,E2 -15403.292} C_VEL
LIN {X 0,Y 322.586,Z 492.536,A -85,B 0,C 180,E1 -15405.479,E2 -15405.479} C_VEL
LIN {X 0,Y 324.227,Z 483.772,A -85,B 0,C 180,E1 -15407.666,E2 -15407.666} C_VEL
LIN {X 0,Y 326.11,Z 474.583,A -85,B 0,C 180,E1 -15409.515,E2 -15409.515} C_VEL
LIN {X 0,Y 328.037,Z 464.431,A -85,B 0,C 180,E1 -15411.195,E2 -15411.195} C_VEL
LIN {X 0,Y 330.073,Z 453.273,A -85,B 0,C 180,E1 -15412.701,E2 -15412.701} C_VEL
LIN {X 0,Y 331.947,Z 440.977,A -85,B 0,C 180,E1 -15414.053,E2 -15414.053} C_VEL
LIN {X 0,Y 333.337,Z 429.113,A -85,B 0,C 180,E1 -15415.114,E2 -15415.114} C_VEL
LIN {X 0,Y 330.535,Z 415.52,A -85,B 0,C 180,E1 -15416.438,E2 -15416.438} C_VEL
LIN {X 0,Y 326.43,Z 401.075,A -85,B 0,C 180,E1 -15417.678,E2 -15417.678} C_VEL
LIN {X 0,Y 321.324,Z 387.153,A -85,B 0,C 180,E1 -15418.75,E2 -15418.75} C_VEL
LIN {X 0,Y 319.82,Z 382.953,A -85,B 0,C 180,E1 -15419.029,E2 -15419.029} C_VEL
LIN {X 0,Y 319.824,Z 381.974,A -85,B 0,C 180,E1 -15419.632,E2 -15419.632} C_VEL
LIN {X 0,Y 320.277,Z 377.193,A -85,B 0,C 180,E1 -15423.503,E2 -15423.503} C_VEL
LIN {X 0,Y 320.598,Z 373.91,A -85,B 0,C 180,E1 -15426.291,E2 -15426.291} C_VEL
LIN {X 0,Y 320.789,Z 370.338,A -85,B 0,C 180,E1 -15429.446,E2 -15429.446} C_VEL
LIN {X 0,Y 320.441,Z 366.804,A -85,B 0,C 180,E1 -15432.836,E2 -15432.836} C_VEL
LIN {X 0,Y 319.88,Z 363.247,A -85,B 0,C 180,E1 -15436.472,E2 -15436.472} C_VEL
LIN {X 0,Y 319.531,Z 361.304,A -85,B 0,C 180,E1 -15438.712,E2 -15438.712} C_VEL
LIN {X 0,Y 319.565,Z 361.302,A -85,B 0,C 180,E1 -15442.348,E2 -15442.348} C_VEL
LIN {X 0,Y 319.564,Z 361.305,A -85,B 0,C 180,E1 -15445.124,E2 -15445.124} C_VEL
LIN {X 0,Y 319.533,Z 361.306,A -85,B 0,C 180,E1 -15447.407,E2 -15447.407} C_VEL
LIN {X 0,Y 318.851,Z 361.395,A -85,B 0,C 180,E1 -15448.459,E2 -15448.459} C_VEL
LIN {X 0,Y 316.006,Z 361.748,A -85,B 0,C 180,E1 -15450.173,E2 -15450.173} C_VEL
LIN {X 0,Y 313.62,Z 362.043,A -85,B 0,C 180,E1 -15451.563,E2 -15451.563} C_VEL
LIN {X 0,Y 312.618,Z 362.17,A -85,B 0,C 180,E1 -15452.638,E2 -15452.638} C_VEL
LIN {X 0,Y 312.547,Z 362.175,A -85,B 0,C 180,E1 -15453.002,E2 -15453.002} C_VEL
LIN {X 0,Y 312.548,Z 362.176,A -85,B 0,C 180,E1 -15456.124,E2 -15456.124} C_VEL
LIN {X 0,Y 312.558,Z 362.172,A -85,B 0,C 180,E1 -15458.914,E2 -15458.914} C_VEL
LIN {X 0,Y 312.643,Z 362.162,A -85,B 0,C 180,E1 -15461.656,E2 -15461.656} C_VEL
LIN {X 0,Y 312.698,Z 362.157,A -85,B 0,C 180,E1 -15465.686,E2 -15465.686} C_VEL
LIN {X 0,Y 312.707,Z 362.158,A -85,B 0,C 180,E1 -15469.642,E2 -15469.642} C_VEL
LIN {X 0,Y 312.877,Z 362.135,A -85,B 0,C 180,E1 -15472.254,E2 -15472.254} C_VEL
LIN {X 0,Y 312.723,Z 362.151,A -85,B 0,C 180,E1 -15474.842,E2 -15474.842} C_VEL
LIN {X 0,Y 312.994,Z 362.118,A -85,B 0,C 180,E1 -15478.713,E2 -15478.713} C_VEL
LIN {X 0,Y 312.994,Z 362.117,A -85,B 0,C 180,E1 -15481.286,E2 -15481.286} C_VEL
LIN {X 0,Y 312.717,Z 362.152,A -85,B 0,C 180,E1 -15485.157,E2 -15485.157} C_VEL
LIN {X 0,Y 312.897,Z 362.136,A -85,B 0,C 180,E1 -15486.448,E2 -15486.448} C_VEL
LIN {X 0,Y 312.703,Z 362.157,A -85,B 0,C 180,E1 -15490.358,E2 -15490.358} C_VEL
LIN {X 0,Y 312.704,Z 362.161,A -85,B 0,C 180,E1 -15494.888,E2 -15494.888} C_VEL
LIN {X 0,Y 312.635,Z 362.17,A -85,B 0,C 180,E1 -15499.237,E2 -15499.237} C_VEL
LIN {X 0,Y 312.549,Z 362.176,A -85,B 0,C 180,E1 -15502.789,E2 -15502.789} C_VEL
LIN {X 0,Y 312.606,Z 362.171,A -85,B 0,C 180,E1 -15505.935,E2 -15505.935} C_VEL
LIN {X 0,Y 312.548,Z 362.175,A -85,B 0,C 180,E1 -15509.649,E2 -15509.649} C_VEL
LIN {X 0,Y 312.522,Z 362.184,A -85,B 0,C 180,E1 -15513.688,E2 -15513.688} C_VEL
LIN {X 0,Y 312.554,Z 362.394,A -85,B 0,C 180,E1 -15515.776,E2 -15515.776} C_VEL
LIN {X 0,Y 313.316,Z 366.103,A -85,B 0,C 180,E1 -15518.908,E2 -15518.908} C_VEL
LIN {X 0,Y 314.238,Z 370.661,A -85,B 0,C 180,E1 -15522.434,E2 -15522.434} C_VEL
LIN {X 0,Y 315.275,Z 376.044,A -85,B 0,C 180,E1 -15526.287,E2 -15526.287} C_VEL
LIN {X 0,Y 316.283,Z 381.521,A -85,B 0,C 180,E1 -15529.879,E2 -15529.879} C_VEL
LIN {X 0,Y 317.03,Z 386.456,A -85,B 0,C 180,E1 -15532.945,E2 -15532.945} C_VEL
LIN {X 0,Y 316.634,Z 389.65,A -85,B 0,C 180,E1 -15534.753,E2 -15534.753} C_VEL
LIN {X 0,Y 315.484,Z 395.212,A -85,B 0,C 180,E1 -15537.835,E2 -15537.835} C_VEL
LIN {X 0,Y 320.414,Z 412.784,A -85,B 0,C 180,E1 -15538.989,E2 -15538.989} C_VEL
LIN {X 0,Y 323.604,Z 427.502,A -85,B 0,C 180,E1 -15540.113,E2 -15540.113} C_VEL
LIN {X 0,Y 325.678,Z 441.252,A -85,B 0,C 180,E1 -15541.312,E2 -15541.312} C_VEL
LIN {X 0,Y 326.395,Z 448.255,A -85,B 0,C 180,E1 -15541.984,E2 -15541.984} C_VEL
LIN {X 0,Y 324.645,Z 460.955,A -85,B 0,C 180,E1 -15543.133,E2 -15543.133} C_VEL
LIN {X 0,Y 322.255,Z 474.769,A -85,B 0,C 180,E1 -15544.659,E2 -15544.659} C_VEL
LIN {X 0,Y 320.168,Z 486.186,A -85,B 0,C 180,E1 -15546.212,E2 -15546.212} C_VEL
LIN {X 0,Y 318.099,Z 496.822,A -85,B 0,C 180,E1 -15547.939,E2 -15547.939} C_VEL
LIN {X 0,Y 316.317,Z 506.676,A -85,B 0,C 180,E1 -15549.856,E2 -15549.856} C_VEL
LIN {X 0,Y 314.39,Z 516.323,A -85,B 0,C 180,E1 -15552.099,E2 -15552.099} C_VEL
LIN {X 0,Y 313.037,Z 524.354,A -85,B 0,C 180,E1 -15554.37,E2 -15554.37} C_VEL
LIN {X 0,Y 311.878,Z 531.836,A -85,B 0,C 180,E1 -15556.977,E2 -15556.977} C_VEL
LIN {X 0,Y 311.155,Z 537.743,A -85,B 0,C 180,E1 -15559.59,E2 -15559.59} C_VEL
LIN {X 0,Y 310.881,Z 542.233,A -85,B 0,C 180,E1 -15562.204,E2 -15562.204} C_VEL
LIN {X 0,Y 310.742,Z 545.391,A -85,B 0,C 180,E1 -15564.809,E2 -15564.809} C_VEL
LIN {X 0,Y 310.751,Z 547.278,A -85,B 0,C 180,E1 -15567.407,E2 -15567.407} C_VEL
LIN {X 0,Y 310.854,Z 547.922,A -85,B 0,C 180,E1 -15570,E2 -15570} C_VEL
LIN {X 0,Y 310.752,Z 547.27,A -85,B 0,C 180,E1 -15572.592,E2 -15572.592} C_VEL
LIN {X 0,Y 310.771,Z 545.372,A -85,B 0,C 180,E1 -15575.19,E2 -15575.19} C_VEL
LIN {X 0,Y 310.881,Z 542.209,A -85,B 0,C 180,E1 -15577.796,E2 -15577.796} C_VEL
LIN {X 0,Y 311.154,Z 537.714,A -85,B 0,C 180,E1 -15580.41,E2 -15580.41} C_VEL
LIN {X 0,Y 311.869,Z 531.792,A -85,B 0,C 180,E1 -15583.023,E2 -15583.023} C_VEL
LIN {X 0,Y 313.035,Z 524.293,A -85,B 0,C 180,E1 -15585.629,E2 -15585.629} C_VEL
LIN {X 0,Y 314.385,Z 516.253,A -85,B 0,C 180,E1 -15587.901,E2 -15587.901} C_VEL
LIN {X 0,Y 316.265,Z 506.591,A -85,B 0,C 180,E1 -15590.148,E2 -15590.148} C_VEL
LIN {X 0,Y 318.107,Z 496.722,A -85,B 0,C 180,E1 -15592.061,E2 -15592.061} C_VEL
LIN {X 0,Y 320.282,Z 484.99,A -85,B 0,C 180,E1 -15593.951,E2 -15593.951} C_VEL
LIN {X 0,Y 322.648,Z 472.041,A -85,B 0,C 180,E1 -15595.653,E2 -15595.653} C_VEL
LIN {X 0,Y 324.89,Z 459.194,A -85,B 0,C 180,E1 -15597.018,E2 -15597.018} C_VEL
LIN {X 0,Y 326.383,Z 448.073,A -85,B 0,C 180,E1 -15598.012,E2 -15598.012} C_VEL
LIN {X 0,Y 324.85,Z 435.401,A -85,B 0,C 180,E1 -15599.2,E2 -15599.2} C_VEL
LIN {X 0,Y 322.306,Z 420.965,A -85,B 0,C 180,E1 -15600.381,E2 -15600.381} C_VEL
LIN {X 0,Y 318.689,Z 406.418,A -85,B 0,C 180,E1 -15601.427,E2 -15601.427} C_VEL
LIN {X 0,Y 315.449,Z 395.186,A -85,B 0,C 180,E1 -15602.155,E2 -15602.155} C_VEL
LIN {X 0,Y 316.619,Z 389.61,A -85,B 0,C 180,E1 -15605.249,E2 -15605.249} C_VEL
LIN {X 0,Y 317.024,Z 386.422,A -85,B 0,C 180,E1 -15607.054,E2 -15607.054} C_VEL
LIN {X 0,Y 316.25,Z 381.464,A -85,B 0,C 180,E1 -15610.126,E2 -15610.126} C_VEL
LIN {X 0,Y 315.267,Z 376.002,A -85,B 0,C 180,E1 -15613.714,E2 -15613.714} C_VEL
LIN {X 0,Y 314.225,Z 370.586,A -85,B 0,C 180,E1 -15617.569,E2 -15617.569} C_VEL
LIN {X 0,Y 313.319,Z 366.045,A -85,B 0,C 180,E1 -15621.093,E2 -15621.093} C_VEL
LIN {X 0,Y 312.534,Z 362.186,A -85,B 0,C 180,E1 -15624.419,E2 -15624.419} C_VEL
LIN {X 0,Y 312.506,Z 362.19,A -85,B 0,C 180,E1 -15627.334,E2 -15627.334} C_VEL
LIN {X 0,Y 312.554,Z 362.182,A -85,B 0,C 180,E1 -15631.276,E2 -15631.276} C_VEL
LIN {X 0,Y 312.588,Z 362.172,A -85,B 0,C 180,E1 -15634.711,E2 -15634.711} C_VEL
LIN {X 0,Y 312.589,Z 362.173,A -85,B 0,C 180,E1 -15637.529,E2 -15637.529} C_VEL
LIN {X 0,Y 312.641,Z 362.162,A -85,B 0,C 180,E1 -15641.657,E2 -15641.657} C_VEL
LIN {X 0,Y 312.697,Z 362.158,A -85,B 0,C 180,E1 -15645.687,E2 -15645.687} C_VEL
LIN {X 0,Y 312.702,Z 362.155,A -85,B 0,C 180,E1 -15649.642,E2 -15649.642} C_VEL
LIN {X 0,Y 312.897,Z 362.128,A -85,B 0,C 180,E1 -15653.552,E2 -15653.552} C_VEL
LIN {X 0,Y 312.939,Z 362.123,A -85,B 0,C 180,E1 -15657.426,E2 -15657.426} C_VEL
LIN {X 0,Y 313.105,Z 362.103,A -85,B 0,C 180,E1 -15660,E2 -15660} C_VEL
LIN {X 0,Y 312.939,Z 362.129,A -85,B 0,C 180,E1 -15662.575,E2 -15662.575} C_VEL
LIN {X 0,Y 312.897,Z 362.133,A -85,B 0,C 180,E1 -15666.653,E2 -15666.653} C_VEL
LIN {X 0,Y 312.791,Z 362.147,A -85,B 0,C 180,E1 -15669.049,E2 -15669.049} C_VEL
LIN {X 0,Y 312.641,Z 362.167,A -85,B 0,C 180,E1 -15672.991,E2 -15672.991} C_VEL
LIN {X 0,Y 312.642,Z 362.164,A -85,B 0,C 180,E1 -15675.65,E2 -15675.65} C_VEL
LIN {X 0,Y 312.634,Z 362.167,A -85,B 0,C 180,E1 -15679.237,E2 -15679.237} C_VEL
LIN {X 0,Y 312.549,Z 362.178,A -85,B 0,C 180,E1 -15682.79,E2 -15682.79} C_VEL
LIN {X 0,Y 312.606,Z 362.17,A -85,B 0,C 180,E1 -15685.936,E2 -15685.936} C_VEL
LIN {X 0,Y 312.548,Z 362.173,A -85,B 0,C 180,E1 -15689.65,E2 -15689.65} C_VEL
LIN {X 0,Y 312.522,Z 362.182,A -85,B 0,C 180,E1 -15693.689,E2 -15693.689} C_VEL
LIN {X 0,Y 312.523,Z 362.183,A -85,B 0,C 180,E1 -15697.386,E2 -15697.386} C_VEL
LIN {X 0,Y 312.509,Z 362.371,A -85,B 0,C 180,E1 -15701.066,E2 -15701.066} C_VEL
LIN {X 0,Y 313,Z 365.157,A -85,B 0,C 180,E1 -15704.112,E2 -15704.112} C_VEL
LIN {X 0,Y 313.569,Z 368.637,A -85,B 0,C 180,E1 -15707.748,E2 -15707.748} C_VEL
LIN {X 0,Y 313.759,Z 372.17,A -85,B 0,C 180,E1 -15711.157,E2 -15711.157} C_VEL
LIN {X 0,Y 313.528,Z 375.731,A -85,B 0,C 180,E1 -15714.351,E2 -15714.351} C_VEL
LIN {X 0,Y 313.142,Z 379.324,A -85,B 0,C 180,E1 -15717.408,E2 -15717.408} C_VEL
LIN {X 0,Y 312.835,Z 383.061,A -85,B 0,C 180,E1 -15720.334,E2 -15720.334} C_VEL
LIN {X 0,Y 314.008,Z 386.338,A -85,B 0,C 180,E1 -15720.56,E2 -15720.56} C_VEL
LIN {X 0,Y 319.21,Z 400.275,A -85,B 0,C 180,E1 -15721.667,E2 -15721.667} C_VEL
LIN {X 0,Y 323.124,Z 413.357,A -85,B 0,C 180,E1 -15722.822,E2 -15722.822} C_VEL
LIN {X 0,Y 325.943,Z 425.874,A -85,B 0,C 180,E1 -15724.05,E2 -15724.05} C_VEL
LIN {X 0,Y 326.775,Z 431.092,A -85,B 0,C 180,E1 -15724.596,E2 -15724.596} C_VEL
LIN {X 0,Y 325.124,Z 443.433,A -85,B 0,C 180,E1 -15725.75,E2 -15725.75} C_VEL
LIN {X 0,Y 323.261,Z 455.298,A -85,B 0,C 180,E1 -15727.131,E2 -15727.131} C_VEL
LIN {X 0,Y 321.297,Z 465.181,A -85,B 0,C 180,E1 -15728.507,E2 -15728.507} C_VEL
LIN {X 0,Y 319.164,Z 476.052,A -85,B 0,C 180,E1 -15730.378,E2 -15730.378} C_VEL
LIN {X 0,Y 317.291,Z 485.011,A -85,B 0,C 180,E1 -15732.261,E2 -15732.261} C_VEL
LIN {X 0,Y 315.495,Z 493.626,A -85,B 0,C 180,E1 -15734.496,E2 -15734.496} C_VEL
LIN {X 0,Y 314.126,Z 499.711,A -85,B 0,C 180,E1 -15736.413,E2 -15736.413} C_VEL
LIN {X 0,Y 312.801,Z 506.168,A -85,B 0,C 180,E1 -15738.99,E2 -15738.99} C_VEL
LIN {X 0,Y 311.893,Z 511.041,A -85,B 0,C 180,E1 -15741.578,E2 -15741.578} C_VEL
LIN {X 0,Y 311.479,Z 513.788,A -85,B 0,C 180,E1 -15743.522,E2 -15743.522} C_VEL
LIN {X 0,Y 311.04,Z 516.263,A -85,B 0,C 180,E1 -15746.113,E2 -15746.113} C_VEL
LIN {X 0,Y 310.91,Z 517.489,A -85,B 0,C 180,E1 -15748.705,E2 -15748.705} C_VEL
LIN {X 0,Y 310.91,Z 517.513,A -85,B 0,C 180,E1 -15751.295,E2 -15751.295} C_VEL
LIN {X 0,Y 311.039,Z 516.34,A -85,B 0,C 180,E1 -15753.887,E2 -15753.887} C_VEL
LIN {X 0,Y 311.479,Z 513.92,A -85,B 0,C 180,E1 -15756.478,E2 -15756.478} C_VEL
LIN {X 0,Y 312.071,Z 510.177,A -85,B 0,C 180,E1 -15759.07,E2 -15759.07} C_VEL
LIN {X 0,Y 313.064,Z 504.97,A -85,B 0,C 180,E1 -15761.657,E2 -15761.657} C_VEL
LIN {X 0,Y 314.437,Z 498.12,A -85,B 0,C 180,E1 -15764.233,E2 -15764.233} C_VEL
LIN {X 0,Y 316.244,Z 490.554,A -85,B 0,C 180,E1 -15766.46,E2 -15766.46} C_VEL
LIN {X 0,Y 317.786,Z 482.697,A -85,B 0,C 180,E1 -15768.37,E2 -15768.37} C_VEL
LIN {X 0,Y 319.811,Z 473.224,A -85,B 0,C 180,E1 -15770.25,E2 -15770.25} C_VEL
LIN {X 0,Y 321.815,Z 462.735,A -85,B 0,C 180,E1 -15771.962,E2 -15771.962} C_VEL
LIN {X 0,Y 323.98,Z 451.148,A -85,B 0,C 180,E1 -15773.491,E2 -15773.491} C_VEL
LIN {X 0,Y 325.844,Z 438.754,A -85,B 0,C 180,E1 -15774.823,E2 -15774.823} C_VEL
LIN {X 0,Y 326.766,Z 431.497,A -85,B 0,C 180,E1 -15775.478,E2 -15775.478} C_VEL
LIN {X 0,Y 325.46,Z 423.171,A -85,B 0,C 180,E1 -15776.341,E2 -15776.341} C_VEL
LIN {X 0,Y 322.262,Z 410.093,A -85,B 0,C 180,E1 -15777.594,E2 -15777.594} C_VEL
LIN {X 0,Y 317.885,Z 396.249,A -85,B 0,C 180,E1 -15778.779,E2 -15778.779} C_VEL
LIN {X 0,Y 312.964,Z 383.614,A -85,B 0,C 180,E1 -15779.752,E2 -15779.752} C_VEL
LIN {X 0,Y 312.836,Z 382.871,A -85,B 0,C 180,E1 -15779.809,E2 -15779.809} C_VEL
LIN {X 0,Y 313.319,Z 377.68,A -85,B 0,C 180,E1 -15784.11,E2 -15784.11} C_VEL
LIN {X 0,Y 313.656,Z 374.111,A -85,B 0,C 180,E1 -15787.228,E2 -15787.228} C_VEL
LIN {X 0,Y 313.767,Z 372.319,A -85,B 0,C 180,E1 -15788.842,E2 -15788.842} C_VEL
LIN {X 0,Y 313.534,Z 368.75,A -85,B 0,C 180,E1 -15792.258,E2 -15792.258} C_VEL
LIN {X 0,Y 313.023,Z 365.227,A -85,B 0,C 180,E1 -15795.928,E2 -15795.928} C_VEL
LIN {X 0,Y 312.469,Z 362.183,A -85,B 0,C 180,E1 -15799.287,E2 -15799.287} C_VEL
LIN {X 0,Y 312.529,Z 362.179,A -85,B 0,C 180,E1 -15802.615,E2 -15802.615} C_VEL
LIN {X 0,Y 312.523,Z 362.181,A -85,B 0,C 180,E1 -15806.311,E2 -15806.311} C_VEL
LIN {X 0,Y 312.549,Z 362.18,A -85,B 0,C 180,E1 -15810.35,E2 -15810.35} C_VEL
LIN {X 0,Y 312.547,Z 362.175,A -85,B 0,C 180,E1 -15813.002,E2 -15813.002} C_VEL
LIN {X 0,Y 311.91,Z 362.26,A -85,B 0,C 180,E1 -15814.077,E2 -15814.077} C_VEL
LIN {X 0,Y 309.068,Z 362.617,A -85,B 0,C 180,E1 -15815.827,E2 -15815.827} C_VEL
LIN {X 0,Y 306.635,Z 362.917,A -85,B 0,C 180,E1 -15817.246,E2 -15817.246} C_VEL
LIN {X 0,Y 305.582,Z 363.044,A -85,B 0,C 180,E1 -15818.345,E2 -15818.345} C_VEL
LIN {X 0,Y 305.493,Z 363.052,A -85,B 0,C 180,E1 -15818.718,E2 -15818.718} C_VEL
LIN {X 0,Y 305.594,Z 363.043,A -85,B 0,C 180,E1 -15821.218,E2 -15821.218} C_VEL
LIN {X 0,Y 305.653,Z 363.033,A -85,B 0,C 180,E1 -15825.349,E2 -15825.349} C_VEL
LIN {X 0,Y 305.644,Z 363.037,A -85,B 0,C 180,E1 -15829.4,E2 -15829.4} C_VEL
LIN {X 0,Y 305.818,Z 363.012,A -85,B 0,C 180,E1 -15832.074,E2 -15832.074} C_VEL
LIN {X 0,Y 305.694,Z 363.026,A -85,B 0,C 180,E1 -15834.723,E2 -15834.723} C_VEL
LIN {X 0,Y 305.96,Z 362.994,A -85,B 0,C 180,E1 -15838.684,E2 -15838.684} C_VEL
LIN {X 0,Y 305.96,Z 362.993,A -85,B 0,C 180,E1 -15841.316,E2 -15841.316} C_VEL
LIN {X 0,Y 305.687,Z 363.028,A -85,B 0,C 180,E1 -15845.276,E2 -15845.276} C_VEL
LIN {X 0,Y 305.776,Z 363.017,A -85,B 0,C 180,E1 -15847.926,E2 -15847.926} C_VEL
LIN {X 0,Y 305.611,Z 363.043,A -85,B 0,C 180,E1 -15851.945,E2 -15851.945} C_VEL
LIN {X 0,Y 305.642,Z 363.041,A -85,B 0,C 180,E1 -15855.035,E2 -15855.035} C_VEL
LIN {X 0,Y 305.581,Z 363.047,A -85,B 0,C 180,E1 -15859.445,E2 -15859.445} C_VEL
LIN {X 0,Y 305.494,Z 363.056,A -85,B 0,C 180,E1 -15863.041,E2 -15863.041} C_VEL
LIN {X 0,Y 305.551,Z 363.051,A -85,B 0,C 180,E1 -15866.227,E2 -15866.227} C_VEL
LIN {X 0,Y 305.499,Z 363.057,A -85,B 0,C 180,E1 -15869.05,E2 -15869.05} C_VEL
LIN {X 0,Y 305.447,Z 363.062,A -85,B 0,C 180,E1 -15871.951,E2 -15871.951} C_VEL
LIN {X 0,Y 305.482,Z 363.136,A -85,B 0,C 180,E1 -15874.678,E2 -15874.678} C_VEL
LIN {X 0,Y 306.311,Z 367.177,A -85,B 0,C 180,E1 -15878.278,E2 -15878.278} C_VEL
LIN {X 0,Y 307.139,Z 371.249,A -85,B 0,C 180,E1 -15881.573,E2 -15881.573} C_VEL
LIN {X 0,Y 308.014,Z 375.926,A -85,B 0,C 180,E1 -15885.018,E2 -15885.018} C_VEL
LIN {X 0,Y 309.013,Z 381.292,A -85,B 0,C 180,E1 -15888.733,E2 -15888.733} C_VEL
LIN {X 0,Y 310.015,Z 387.132,A -85,B 0,C 180,E1 -15892.508,E2 -15892.508} C_VEL
LIN {X 0,Y 309.949,Z 389.418,A -85,B 0,C 180,E1 -15893.875,E2 -15893.875} C_VEL
LIN {X 0,Y 308.707,Z 395.06,A -85,B 0,C 180,E1 -15897.086,E2 -15897.086} C_VEL
LIN {X 0,Y 313.591,Z 412.164,A -85,B 0,C 180,E1 -15898.256,E2 -15898.256} C_VEL
LIN {X 0,Y 316.777,Z 426.554,A -85,B 0,C 180,E1 -15899.392,E2 -15899.392} C_VEL
LIN {X 0,Y 318.771,Z 439.125,A -85,B 0,C 180,E1 -15900.513,E2 -15900.513} C_VEL
LIN {X 0,Y 319.87,Z 449.229,A -85,B 0,C 180,E1 -15901.505,E2 -15901.505} C_VEL
LIN {X 0,Y 318.031,Z 462.034,A -85,B 0,C 180,E1 -15902.706,E2 -15902.706} C_VEL
LIN {X 0,Y 315.559,Z 475.578,A -85,B 0,C 180,E1 -15904.259,E2 -15904.259} C_VEL
LIN {X 0,Y 313.402,Z 486.841,A -85,B 0,C 180,E1 -15905.842,E2 -15905.842} C_VEL
LIN {X 0,Y 311.194,Z 497.721,A -85,B 0,C 180,E1 -15907.675,E2 -15907.675} C_VEL
LIN {X 0,Y 309.288,Z 507.803,A -85,B 0,C 180,E1 -15909.725,E2 -15909.725} C_VEL
LIN {X 0,Y 307.321,Z 517.21,A -85,B 0,C 180,E1 -15912.017,E2 -15912.017} C_VEL
LIN {X 0,Y 305.936,Z 525.091,A -85,B 0,C 180,E1 -15914.362,E2 -15914.362} C_VEL
LIN {X 0,Y 304.874,Z 531.478,A -85,B 0,C 180,E1 -15916.672,E2 -15916.672} C_VEL
LIN {X 0,Y 304.099,Z 537.39,A -85,B 0,C 180,E1 -15919.345,E2 -15919.345} C_VEL
LIN {X 0,Y 303.804,Z 541.884,A -85,B 0,C 180,E1 -15922.021,E2 -15922.021} C_VEL
LIN {X 0,Y 303.665,Z 545.044,A -85,B 0,C 180,E1 -15924.688,E2 -15924.688} C_VEL
LIN {X 0,Y 303.672,Z 546.934,A -85,B 0,C 180,E1 -15927.347,E2 -15927.347} C_VEL
LIN {X 0,Y 303.762,Z 547.576,A -85,B 0,C 180,E1 -15930,E2 -15930} C_VEL
LIN {X 0,Y 303.674,Z 546.925,A -85,B 0,C 180,E1 -15932.653,E2 -15932.653} C_VEL
LIN {X 0,Y 303.684,Z 545.025,A -85,B 0,C 180,E1 -15935.311,E2 -15935.311} C_VEL
LIN {X 0,Y 303.804,Z 541.858,A -85,B 0,C 180,E1 -15937.978,E2 -15937.978} C_VEL
LIN {X 0,Y 304.099,Z 537.359,A -85,B 0,C 180,E1 -15940.654,E2 -15940.654} C_VEL
LIN {X 0,Y 304.866,Z 531.432,A -85,B 0,C 180,E1 -15943.328,E2 -15943.328} C_VEL
LIN {X 0,Y 306.117,Z 523.927,A -85,B 0,C 180,E1 -15945.992,E2 -15945.992} C_VEL
LIN {X 0,Y 307.54,Z 515.876,A -85,B 0,C 180,E1 -15948.314,E2 -15948.314} C_VEL
LIN {X 0,Y 309.533,Z 506.204,A -85,B 0,C 180,E1 -15950.605,E2 -15950.605} C_VEL
LIN {X 0,Y 311.45,Z 496.317,A -85,B 0,C 180,E1 -15952.558,E2 -15952.558} C_VEL
LIN {X 0,Y 313.697,Z 484.561,A -85,B 0,C 180,E1 -15954.486,E2 -15954.486} C_VEL
LIN {X 0,Y 316.216,Z 471.583,A -85,B 0,C 180,E1 -15956.214,E2 -15956.214} C_VEL
LIN {X 0,Y 318.544,Z 458.692,A -85,B 0,C 180,E1 -15957.602,E2 -15957.602} C_VEL
LIN {X 0,Y 319.847,Z 449.094,A -85,B 0,C 180,E1 -15958.488,E2 -15958.488} C_VEL
LIN {X 0,Y 318.133,Z 434.732,A -85,B 0,C 180,E1 -15959.878,E2 -15959.878} C_VEL
LIN {X 0,Y 315.51,Z 420.121,A -85,B 0,C 180,E1 -15961.107,E2 -15961.107} C_VEL
LIN {X 0,Y 311.452,Z 404.495,A -85,B 0,C 180,E1 -15962.271,E2 -15962.271} C_VEL
LIN {X 0,Y 308.697,Z 395.019,A -85,B 0,C 180,E1 -15962.91,E2 -15962.91} C_VEL
LIN {X 0,Y 309.892,Z 389.374,A -85,B 0,C 180,E1 -15966.132,E2 -15966.132} C_VEL
LIN {X 0,Y 309.962,Z 386.666,A -85,B 0,C 180,E1 -15967.748,E2 -15967.748} C_VEL
LIN {X 0,Y 308.98,Z 381.098,A -85,B 0,C 180,E1 -15971.357,E2 -15971.357} C_VEL
LIN {X 0,Y 308.002,Z 375.808,A -85,B 0,C 180,E1 -15975.021,E2 -15975.021} C_VEL
LIN {X 0,Y 306.948,Z 370.39,A -85,B 0,C 180,E1 -15979.076,E2 -15979.076} C_VEL
LIN {X 0,Y 306.329,Z 367.163,A -85,B 0,C 180,E1 -15981.724,E2 -15981.724} C_VEL
LIN {X 0,Y 305.491,Z 363.064,A -85,B 0,C 180,E1 -15985.467,E2 -15985.467} C_VEL
LIN {X 0,Y 305.465,Z 363.064,A -85,B 0,C 180,E1 -15989.591,E2 -15989.591} C_VEL
LIN {X 0,Y 305.536,Z 363.051,A -85,B 0,C 180,E1 -15992.61,E2 -15992.61} C_VEL
LIN {X 0,Y 305.51,Z 363.056,A -85,B 0,C 180,E1 -15995.539,E2 -15995.539} C_VEL
LIN {X 0,Y 305.522,Z 363.053,A -85,B 0,C 180,E1 -15999.815,E2 -15999.815} C_VEL
LIN {X 0,Y 305.578,Z 363.045,A -85,B 0,C 180,E1 -16002.603,E2 -16002.603} C_VEL
LIN {X 0,Y 305.652,Z 363.036,A -85,B 0,C 180,E1 -16005.349,E2 -16005.349} C_VEL
LIN {X 0,Y 305.64,Z 363.037,A -85,B 0,C 180,E1 -16009.4,E2 -16009.4} C_VEL
LIN {X 0,Y 305.776,Z 363.022,A -85,B 0,C 180,E1 -16012.074,E2 -16012.074} C_VEL
LIN {X 0,Y 305.688,Z 363.031,A -85,B 0,C 180,E1 -16014.724,E2 -16014.724} C_VEL
LIN {X 0,Y 305.961,Z 362.999,A -85,B 0,C 180,E1 -16018.684,E2 -16018.684} C_VEL
LIN {X 0,Y 305.959,Z 362.993,A -85,B 0,C 180,E1 -16021.316,E2 -16021.316} C_VEL
LIN {X 0,Y 305.856,Z 363.011,A -85,B 0,C 180,E1 -16026.598,E2 -16026.598} C_VEL
LIN {X 0,Y 305.739,Z 363.026,A -85,B 0,C 180,E1 -16029.26,E2 -16029.26} C_VEL
LIN {X 0,Y 305.595,Z 363.046,A -85,B 0,C 180,E1 -16033.296,E2 -16033.296} C_VEL
LIN {X 0,Y 305.597,Z 363.043,A -85,B 0,C 180,E1 -16036.02,E2 -16036.02} C_VEL
LIN {X 0,Y 305.58,Z 363.046,A -85,B 0,C 180,E1 -16039.445,E2 -16039.445} C_VEL
LIN {X 0,Y 305.494,Z 363.058,A -85,B 0,C 180,E1 -16043.042,E2 -16043.042} C_VEL
LIN {X 0,Y 305.551,Z 363.048,A -85,B 0,C 180,E1 -16046.227,E2 -16046.227} C_VEL
LIN {X 0,Y 305.498,Z 363.053,A -85,B 0,C 180,E1 -16049.05,E2 -16049.05} C_VEL
LIN {X 0,Y 305.447,Z 363.064,A -85,B 0,C 180,E1 -16051.952,E2 -16051.952} C_VEL
LIN {X 0,Y 305.465,Z 363.061,A -85,B 0,C 180,E1 -16055.113,E2 -16055.113} C_VEL
LIN {X 0,Y 305.468,Z 363.062,A -85,B 0,C 180,E1 -16059.255,E2 -16059.255} C_VEL
LIN {X 0,Y 305.464,Z 363.063,A -85,B 0,C 180,E1 -16060.107,E2 -16060.107} C_VEL
LIN {X 0,Y 305.943,Z 366.089,A -85,B 0,C 180,E1 -16063.563,E2 -16063.563} C_VEL
LIN {X 0,Y 306.495,Z 369.498,A -85,B 0,C 180,E1 -16067.204,E2 -16067.204} C_VEL
LIN {X 0,Y 306.729,Z 372.38,A -85,B 0,C 180,E1 -16070.092,E2 -16070.092} C_VEL
LIN {X 0,Y 306.744,Z 374.162,A -85,B 0,C 180,E1 -16071.785,E2 -16071.785} C_VEL
LIN {X 0,Y 306.342,Z 378.507,A -85,B 0,C 180,E1 -16075.68,E2 -16075.68} C_VEL
LIN {X 0,Y 305.888,Z 383.122,A -85,B 0,C 180,E1 -16079.543,E2 -16079.543} C_VEL
LIN {X 0,Y 307.038,Z 386.416,A -85,B 0,C 180,E1 -16079.778,E2 -16079.778} C_VEL
LIN {X 0,Y 312.338,Z 400.265,A -85,B 0,C 180,E1 -16080.935,E2 -16080.935} C_VEL
LIN {X 0,Y 316.162,Z 412.821,A -85,B 0,C 180,E1 -16082.083,E2 -16082.083} C_VEL
LIN {X 0,Y 319.048,Z 425.215,A -85,B 0,C 180,E1 -16083.332,E2 -16083.332} C_VEL
LIN {X 0,Y 320.297,Z 432.296,A -85,B 0,C 180,E1 -16084.11,E2 -16084.11} C_VEL
LIN {X 0,Y 318.477,Z 445.341,A -85,B 0,C 180,E1 -16085.385,E2 -16085.385} C_VEL
LIN {X 0,Y 316.508,Z 456.909,A -85,B 0,C 180,E1 -16086.788,E2 -16086.788} C_VEL
LIN {X 0,Y 314.374,Z 467.523,A -85,B 0,C 180,E1 -16088.354,E2 -16088.354} C_VEL
LIN {X 0,Y 312.129,Z 478.049,A -85,B 0,C 180,E1 -16090.26,E2 -16090.26} C_VEL
LIN {X 0,Y 310.438,Z 485.792,A -85,B 0,C 180,E1 -16091.96,E2 -16091.96} C_VEL
LIN {X 0,Y 308.662,Z 493.991,A -85,B 0,C 180,E1 -16094.143,E2 -16094.143} C_VEL
LIN {X 0,Y 307.225,Z 500.068,A -85,B 0,C 180,E1 -16096.102,E2 -16096.102} C_VEL
LIN {X 0,Y 305.841,Z 506.519,A -85,B 0,C 180,E1 -16098.736,E2 -16098.736} C_VEL
LIN {X 0,Y 304.868,Z 511.39,A -85,B 0,C 180,E1 -16101.382,E2 -16101.382} C_VEL
LIN {X 0,Y 304.418,Z 514.136,A -85,B 0,C 180,E1 -16103.371,E2 -16103.371} C_VEL
LIN {X 0,Y 303.977,Z 516.608,A -85,B 0,C 180,E1 -16106.023,E2 -16106.023} C_VEL
LIN {X 0,Y 303.819,Z 517.835,A -85,B 0,C 180,E1 -16108.675,E2 -16108.675} C_VEL
LIN {X 0,Y 303.819,Z 517.859,A -85,B 0,C 180,E1 -16111.326,E2 -16111.326} C_VEL
LIN {X 0,Y 303.976,Z 516.685,A -85,B 0,C 180,E1 -16113.977,E2 -16113.977} C_VEL
LIN {X 0,Y 304.418,Z 514.266,A -85,B 0,C 180,E1 -16116.629,E2 -16116.629} C_VEL
LIN {X 0,Y 305.048,Z 510.526,A -85,B 0,C 180,E1 -16119.281,E2 -16119.281} C_VEL
LIN {X 0,Y 306.122,Z 505.321,A -85,B 0,C 180,E1 -16121.925,E2 -16121.925} C_VEL
LIN {X 0,Y 307.56,Z 498.477,A -85,B 0,C 180,E1 -16124.558,E2 -16124.558} C_VEL
LIN {X 0,Y 309.434,Z 490.92,A -85,B 0,C 180,E1 -16126.833,E2 -16126.833} C_VEL
LIN {X 0,Y 311.049,Z 483.074,A -85,B 0,C 180,E1 -16128.783,E2 -16128.783} C_VEL
LIN {X 0,Y 313.172,Z 473.616,A -85,B 0,C 180,E1 -16130.699,E2 -16130.699} C_VEL
LIN {X 0,Y 315.253,Z 463.15,A -85,B 0,C 180,E1 -16132.444,E2 -16132.444} C_VEL
LIN {X 0,Y 317.508,Z 451.594,A -85,B 0,C 180,E1 -16134,E2 -16134} C_VEL
LIN {X 0,Y 319.392,Z 439.622,A -85,B 0,C 180,E1 -16135.318,E2 -16135.318} C_VEL
LIN {X 0,Y 320.287,Z 432.031,A -85,B 0,C 180,E1 -16136.031,E2 -16136.031} C_VEL
LIN {X 0,Y 317.779,Z 419.014,A -85,B 0,C 180,E1 -16137.417,E2 -16137.417} C_VEL
LIN {X 0,Y 313.85,Z 404.761,A -85,B 0,C 180,E1 -16138.78,E2 -16138.78} C_VEL
LIN {X 0,Y 309.122,Z 391.56,A -85,B 0,C 180,E1 -16139.925,E2 -16139.925} C_VEL
LIN {X 0,Y 306.011,Z 383.718,A -85,B 0,C 180,E1 -16140.543,E2 -16140.543} C_VEL
LIN {X 0,Y 305.915,Z 383.058,A -85,B 0,C 180,E1 -16140.599,E2 -16140.599} C_VEL
LIN {X 0,Y 306.42,Z 377.897,A -85,B 0,C 180,E1 -16144.988,E2 -16144.988} C_VEL
LIN {X 0,Y 306.758,Z 374.318,A -85,B 0,C 180,E1 -16148.213,E2 -16148.213} C_VEL
LIN {X 0,Y 306.616,Z 370.738,A -85,B 0,C 180,E1 -16151.661,E2 -16151.661} C_VEL
LIN {X 0,Y 306.13,Z 367.206,A -85,B 0,C 180,E1 -16155.373,E2 -16155.373} C_VEL
LIN {X 0,Y 305.543,Z 363.607,A -85,B 0,C 180,E1 -16159.382,E2 -16159.382} C_VEL
LIN {X 0,Y 305.465,Z 363.056,A -85,B 0,C 180,E1 -16160.319,E2 -16160.319} C_VEL
LIN {X 0,Y 305.485,Z 363.057,A -85,B 0,C 180,E1 -16163.632,E2 -16163.632} C_VEL
LIN {X 0,Y 305.469,Z 363.06,A -85,B 0,C 180,E1 -16166.483,E2 -16166.483} C_VEL
LIN {X 0,Y 305.467,Z 363.058,A -85,B 0,C 180,E1 -16169.591,E2 -16169.591} C_VEL
LIN {X 0,Y 305.52,Z 363.051,A -85,B 0,C 180,E1 -16173.003,E2 -16173.003} C_VEL
LIN {X 0,Y 305.513,Z 363.054,A -85,B 0,C 180,E1 -16175.539,E2 -16175.539} C_VEL
LIN {X 0,Y 305.493,Z 363.052,A -85,B 0,C 180,E1 -16178.718,E2 -16178.718} C_VEL
LIN {X 0,Y 304.814,Z 363.14,A -85,B 0,C 180,E1 -16179.819,E2 -16179.819} C_VEL
LIN {X 0,Y 301.972,Z 363.492,A -85,B 0,C 180,E1 -16181.612,E2 -16181.612} C_VEL
LIN {X 0,Y 299.606,Z 363.789,A -85,B 0,C 180,E1 -16183.067,E2 -16183.067} C_VEL
LIN {X 0,Y 298.642,Z 363.909,A -85,B 0,C 180,E1 -16184.193,E2 -16184.193} C_VEL
LIN {X 0,Y 298.59,Z 363.912,A -85,B 0,C 180,E1 -16184.574,E2 -16184.574} C_VEL
LIN {X 0,Y 298.599,Z 363.915,A -85,B 0,C 180,E1 -16189.147,E2 -16189.147} C_VEL
LIN {X 0,Y 298.763,Z 363.89,A -85,B 0,C 180,E1 -16191.886,E2 -16191.886} C_VEL
LIN {X 0,Y 298.665,Z 363.902,A -85,B 0,C 180,E1 -16194.599,E2 -16194.599} C_VEL
LIN {X 0,Y 298.927,Z 363.87,A -85,B 0,C 180,E1 -16198.653,E2 -16198.653} C_VEL
LIN {X 0,Y 298.927,Z 363.869,A -85,B 0,C 180,E1 -16201.347,E2 -16201.347} C_VEL
LIN {X 0,Y 298.78,Z 363.894,A -85,B 0,C 180,E1 -16206.754,E2 -16206.754} C_VEL
LIN {X 0,Y 298.635,Z 363.913,A -85,B 0,C 180,E1 -16209.482,E2 -16209.482} C_VEL
LIN {X 0,Y 298.558,Z 363.921,A -85,B 0,C 180,E1 -16213.615,E2 -16213.615} C_VEL
LIN {X 0,Y 298.553,Z 363.924,A -85,B 0,C 180,E1 -16216.408,E2 -16216.408} C_VEL
LIN {X 0,Y 298.516,Z 363.926,A -85,B 0,C 180,E1 -16219.655,E2 -16219.655} C_VEL
LIN {X 0,Y 298.461,Z 363.936,A -85,B 0,C 180,E1 -16223.597,E2 -16223.597} C_VEL
LIN {X 0,Y 298.492,Z 363.932,A -85,B 0,C 180,E1 -16226.574,E2 -16226.574} C_VEL
LIN {X 0,Y 298.424,Z 363.935,A -85,B 0,C 180,E1 -16229.64,E2 -16229.64} C_VEL
LIN {X 0,Y 298.445,Z 363.959,A -85,B 0,C 180,E1 -16233.6,E2 -16233.6} C_VEL
LIN {X 0,Y 299.28,Z 368.276,A -85,B 0,C 180,E1 -16237.63,E2 -16237.63} C_VEL
LIN {X 0,Y 300.257,Z 372.959,A -85,B 0,C 180,E1 -16241.494,E2 -16241.494} C_VEL
LIN {X 0,Y 301.265,Z 378.353,A -85,B 0,C 180,E1 -16245.584,E2 -16245.584} C_VEL
LIN {X 0,Y 302.255,Z 383.761,A -85,B 0,C 180,E1 -16249.378,E2 -16249.378} C_VEL
LIN {X 0,Y 302.951,Z 387.825,A -85,B 0,C 180,E1 -16252.068,E2 -16252.068} C_VEL
LIN {X 0,Y 302.981,Z 390.489,A -85,B 0,C 180,E1 -16253.72,E2 -16253.72} C_VEL
LIN {X 0,Y 301.987,Z 394.851,A -85,B 0,C 180,E1 -16256.285,E2 -16256.285} C_VEL
LIN {X 0,Y 307.166,Z 412.9,A -85,B 0,C 180,E1 -16257.596,E2 -16257.596} C_VEL
LIN {X 0,Y 310.29,Z 427.058,A -85,B 0,C 180,E1 -16258.763,E2 -16258.763} C_VEL
LIN {X 0,Y 312.445,Z 441.439,A -85,B 0,C 180,E1 -16260.097,E2 -16260.097} C_VEL
LIN {X 0,Y 313.324,Z 450.296,A -85,B 0,C 180,E1 -16261.02,E2 -16261.02} C_VEL
LIN {X 0,Y 311.427,Z 463.021,A -85,B 0,C 180,E1 -16262.261,E2 -16262.261} C_VEL
LIN {X 0,Y 309.122,Z 475.141,A -85,B 0,C 180,E1 -16263.682,E2 -16263.682} C_VEL
LIN {X 0,Y 306.647,Z 487.461,A -85,B 0,C 180,E1 -16265.455,E2 -16265.455} C_VEL
LIN {X 0,Y 304.464,Z 497.758,A -85,B 0,C 180,E1 -16267.24,E2 -16267.24} C_VEL
LIN {X 0,Y 302.24,Z 508.901,A -85,B 0,C 180,E1 -16269.586,E2 -16269.586} C_VEL
LIN {X 0,Y 300.257,Z 518.071,A -85,B 0,C 180,E1 -16271.932,E2 -16271.932} C_VEL
LIN {X 0,Y 298.796,Z 525.898,A -85,B 0,C 180,E1 -16274.376,E2 -16274.376} C_VEL
LIN {X 0,Y 297.682,Z 532.783,A -85,B 0,C 180,E1 -16277.039,E2 -16277.039} C_VEL
LIN {X 0,Y 296.942,Z 538.328,A -85,B 0,C 180,E1 -16279.775,E2 -16279.775} C_VEL
LIN {X 0,Y 296.722,Z 541.534,A -85,B 0,C 180,E1 -16281.83,E2 -16281.83} C_VEL
LIN {X 0,Y 296.599,Z 544.699,A -85,B 0,C 180,E1 -16284.561,E2 -16284.561} C_VEL
LIN {X 0,Y 296.595,Z 546.589,A -85,B 0,C 180,E1 -16287.284,E2 -16287.284} C_VEL
LIN {X 0,Y 296.67,Z 547.231,A -85,B 0,C 180,E1 -16290,E2 -16290} C_VEL
LIN {X 0,Y 296.597,Z 546.58,A -85,B 0,C 180,E1 -16292.716,E2 -16292.716} C_VEL
LIN {X 0,Y 296.629,Z 544.472,A -85,B 0,C 180,E1 -16295.676,E2 -16295.676} C_VEL
LIN {X 0,Y 296.788,Z 540.541,A -85,B 0,C 180,E1 -16298.854,E2 -16298.854} C_VEL
LIN {X 0,Y 297.251,Z 535.702,A -85,B 0,C 180,E1 -16301.594,E2 -16301.594} C_VEL
LIN {X 0,Y 298.148,Z 529.388,A -85,B 0,C 180,E1 -16304.33,E2 -16304.33} C_VEL
LIN {X 0,Y 299.591,Z 521.433,A -85,B 0,C 180,E1 -16307.052,E2 -16307.052} C_VEL
LIN {X 0,Y 301.264,Z 512.951,A -85,B 0,C 180,E1 -16309.416,E2 -16309.416} C_VEL
LIN {X 0,Y 303.432,Z 502.72,A -85,B 0,C 180,E1 -16311.752,E2 -16311.752} C_VEL
LIN {X 0,Y 305.551,Z 492.259,A -85,B 0,C 180,E1 -16313.736,E2 -16313.736} C_VEL
LIN {X 0,Y 307.897,Z 480.888,A -85,B 0,C 180,E1 -16315.521,E2 -16315.521} C_VEL
LIN {X 0,Y 310.32,Z 468.524,A -85,B 0,C 180,E1 -16317.115,E2 -16317.115} C_VEL
LIN {X 0,Y 312.828,Z 454.5,A -85,B 0,C 180,E1 -16318.567,E2 -16318.567} C_VEL
LIN {X 0,Y 313.3,Z 450.158,A -85,B 0,C 180,E1 -16318.972,E2 -16318.972} C_VEL
LIN {X 0,Y 311.703,Z 435.898,A -85,B 0,C 180,E1 -16320.41,E2 -16320.41} C_VEL
LIN {X 0,Y 309.119,Z 421.295,A -85,B 0,C 180,E1 -16321.701,E2 -16321.701} C_VEL
LIN {X 0,Y 305.55,Z 407.142,A -85,B 0,C 180,E1 -16322.816,E2 -16322.816} C_VEL
LIN {X 0,Y 301.94,Z 394.868,A -85,B 0,C 180,E1 -16323.678,E2 -16323.678} C_VEL
LIN {X 0,Y 302.932,Z 390.441,A -85,B 0,C 180,E1 -16326.28,E2 -16326.28} C_VEL
LIN {X 0,Y 302.951,Z 387.784,A -85,B 0,C 180,E1 -16327.932,E2 -16327.932} C_VEL
LIN {X 0,Y 301.929,Z 381.914,A -85,B 0,C 180,E1 -16331.853,E2 -16331.853} C_VEL
LIN {X 0,Y 300.985,Z 376.767,A -85,B 0,C 180,E1 -16335.533,E2 -16335.533} C_VEL
LIN {X 0,Y 300.109,Z 372.272,A -85,B 0,C 180,E1 -16339.027,E2 -16339.027} C_VEL
LIN {X 0,Y 299.144,Z 367.503,A -85,B 0,C 180,E1 -16343.015,E2 -16343.015} C_VEL
LIN {X 0,Y 298.444,Z 363.938,A -85,B 0,C 180,E1 -16346.4,E2 -16346.4} C_VEL
LIN {X 0,Y 298.434,Z 363.938,A -85,B 0,C 180,E1 -16350.615,E2 -16350.615} C_VEL
LIN {X 0,Y 298.494,Z 363.931,A -85,B 0,C 180,E1 -16353.471,E2 -16353.471} C_VEL
LIN {X 0,Y 298.437,Z 363.933,A -85,B 0,C 180,E1 -16356.698,E2 -16356.698} C_VEL
LIN {X 0,Y 298.542,Z 363.92,A -85,B 0,C 180,E1 -16360.757,E2 -16360.757} C_VEL
LIN {X 0,Y 298.596,Z 363.913,A -85,B 0,C 180,E1 -16364.995,E2 -16364.995} C_VEL
LIN {X 0,Y 298.596,Z 363.916,A -85,B 0,C 180,E1 -16369.147,E2 -16369.147} C_VEL
LIN {X 0,Y 298.722,Z 363.901,A -85,B 0,C 180,E1 -16371.885,E2 -16371.885} C_VEL
LIN {X 0,Y 298.658,Z 363.905,A -85,B 0,C 180,E1 -16374.599,E2 -16374.599} C_VEL
LIN {X 0,Y 298.927,Z 363.876,A -85,B 0,C 180,E1 -16378.653,E2 -16378.653} C_VEL
LIN {X 0,Y 298.926,Z 363.869,A -85,B 0,C 180,E1 -16381.347,E2 -16381.347} C_VEL
LIN {X 0,Y 298.802,Z 363.888,A -85,B 0,C 180,E1 -16386.754,E2 -16386.754} C_VEL
LIN {X 0,Y 298.684,Z 363.905,A -85,B 0,C 180,E1 -16389.481,E2 -16389.481} C_VEL
LIN {X 0,Y 298.558,Z 363.92,A -85,B 0,C 180,E1 -16393.615,E2 -16393.615} C_VEL
LIN {X 0,Y 298.552,Z 363.922,A -85,B 0,C 180,E1 -16396.409,E2 -16396.409} C_VEL
LIN {X 0,Y 298.515,Z 363.927,A -85,B 0,C 180,E1 -16399.655,E2 -16399.655} C_VEL
LIN {X 0,Y 298.461,Z 363.928,A -85,B 0,C 180,E1 -16403.598,E2 -16403.598} C_VEL
LIN {X 0,Y 298.492,Z 363.925,A -85,B 0,C 180,E1 -16406.574,E2 -16406.574} C_VEL
LIN {X 0,Y 298.424,Z 363.932,A -85,B 0,C 180,E1 -16409.641,E2 -16409.641} C_VEL
LIN {X 0,Y 298.398,Z 363.94,A -85,B 0,C 180,E1 -16412.8,E2 -16412.8} C_VEL
LIN {X 0,Y 298.447,Z 363.936,A -85,B 0,C 180,E1 -16416.807,E2 -16416.807} C_VEL
LIN {X 0,Y 298.451,Z 364.085,A -85,B 0,C 180,E1 -16419.48,E2 -16419.48} C_VEL
LIN {X 0,Y 298.963,Z 367.256,A -85,B 0,C 180,E1 -16423.218,E2 -16423.218} C_VEL
LIN {X 0,Y 299.466,Z 370.4,A -85,B 0,C 180,E1 -16426.679,E2 -16426.679} C_VEL
LIN {X 0,Y 299.736,Z 372.584,A -85,B 0,C 180,E1 -16428.964,E2 -16428.964} C_VEL
LIN {X 0,Y 299.768,Z 374.376,A -85,B 0,C 180,E1 -16430.727,E2 -16430.727} C_VEL
LIN {X 0,Y 299.505,Z 377.971,A -85,B 0,C 180,E1 -16434.081,E2 -16434.081} C_VEL
LIN {X 0,Y 299.047,Z 382.643,A -85,B 0,C 180,E1 -16438.181,E2 -16438.181} C_VEL
LIN {X 0,Y 298.972,Z 383.287,A -85,B 0,C 180,E1 -16438.716,E2 -16438.716} C_VEL
LIN {X 0,Y 300.06,Z 386.427,A -85,B 0,C 180,E1 -16438.949,E2 -16438.949} C_VEL
LIN {X 0,Y 305.363,Z 399.967,A -85,B 0,C 180,E1 -16440.138,E2 -16440.138} C_VEL
LIN {X 0,Y 309.384,Z 412.896,A -85,B 0,C 180,E1 -16441.368,E2 -16441.368} C_VEL
LIN {X 0,Y 312.495,Z 426.131,A -85,B 0,C 180,E1 -16442.756,E2 -16442.756} C_VEL
LIN {X 0,Y 313.812,Z 433.641,A -85,B 0,C 180,E1 -16443.615,E2 -16443.615} C_VEL
LIN {X 0,Y 312.068,Z 445.818,A -85,B 0,C 180,E1 -16444.844,E2 -16444.844} C_VEL
LIN {X 0,Y 310.025,Z 457.345,A -85,B 0,C 180,E1 -16446.273,E2 -16446.273} C_VEL
LIN {X 0,Y 307.78,Z 467.933,A -85,B 0,C 180,E1 -16447.866,E2 -16447.866} C_VEL
LIN {X 0,Y 305.473,Z 478.438,A -85,B 0,C 180,E1 -16449.812,E2 -16449.812} C_VEL
LIN {X 0,Y 303.559,Z 486.658,A -85,B 0,C 180,E1 -16451.666,E2 -16451.666} C_VEL
LIN {X 0,Y 301.839,Z 494.355,A -85,B 0,C 180,E1 -16453.775,E2 -16453.775} C_VEL
LIN {X 0,Y 300.337,Z 500.425,A -85,B 0,C 180,E1 -16455.777,E2 -16455.777} C_VEL
LIN {X 0,Y 298.876,Z 506.872,A -85,B 0,C 180,E1 -16458.47,E2 -16458.47} C_VEL
LIN {X 0,Y 297.849,Z 511.74,A -85,B 0,C 180,E1 -16461.178,E2 -16461.178} C_VEL
